(* IEC 61131-3 sources: PortalRobot/Portal_robot/Device/application (part 2) *)

(* ---- FB_MACHINE.st ---- *)
FUNCTION_BLOCK FB_MACHINE
VAR_INPUT
	xExecute          : BOOL; // Запуск разрешённой операции обслуживания
    xReset            : BOOL; // Сброс ошибки конкретного станка
	xResetGlobal      : BOOL; // Общий сброс ошибок ячейки
	xGlobalError      : BOOL; // Глобальная ошибка ячейки
	xHmiSetPartLoaded : BOOL; // Ручное подтверждение загруженной детали
    xHmiSetPartEmpty  : BOOL; // Ручное подтверждение пустого патрона
	xHmiEnable        : BOOL; // Импульс включения станка в работу
	xHmiDisable       : BOOL; // Импульс отключения станка от работы
	stChangeRecipe    : ARRAY [0..40] OF ST_MACHINE_RECIPE; // Рецепт смены детали
	stLoadRecipe      : ARRAY [0..40] OF ST_MACHINE_RECIPE; // Рецепт загрузки заготовки
	stUnloadRecipe    : ARRAY [0..40] OF ST_MACHINE_RECIPE; // Рецепт выгрузки детали
	stPoints          : ST_MACHINE_POINTS; // Имена рабочих точек станка
	stRobotStatus     : ST_ROBOT_STATUS; // Статусы робота
	stMachineStatus   : ST_MACHINE_IO_STATUS; // Состояние исполнительных механизмов станка
END_VAR
VAR_OUTPUT
	Command : ST_MACHINE_COMMAND; // Команды станку и роботу
	Status  : ST_MACHINE_PUBLIC; // Публичные статусы станка
	Diag    : ST_MACHINE_DIAG; // Состояние автомата и выбранная операция
	Error   : ST_MACHINE_ERRORS; // Активные и последние ошибки
END_VAR
VAR
	eState                  : E_MACHINE_STATE := E_MACHINE_STATE.DISABLED; // Текущее состояние автомата
	ePartState              : E_PART_STATE := E_PART_STATE.UNKNOWN; // Состояние детали в патроне
	uiIndex                 : UINT; // Индекс команды рецепта
	tofErrorDoor            : TOF; // Контроль закрытия двери при нахождении робота внутри
	rtExectue               : R_TRIG; // Фронт команды запуска
	rtEnabledMachine        : R_TRIG; // Фронт команды включения
	rtDisabledMachine       : R_TRIG; // Фронт команды отключения
	rtCycleDone             : R_TRIG; // Фронт завершения цикла станка
    rtSetPartLoaded         : R_TRIG; // Фронт ручного подтверждения детали
    rtSetPartEmpty          : R_TRIG; // Фронт ручного подтверждения пустого патрона
	xRetreatStarted         : BOOL; // Начат отход робота от станка
	xRobotInsideMachine     : BOOL; // Робот находится внутри рабочей зоны
	xRobotDone              : BOOL; // Робот освобождён алгоритмом станка
	xServiceDoorCloseDemand : BOOL; // Внутренний запрос закрытия двери
	xServiceDoorOpenDemand  : BOOL; // Внутренний запрос открытия двери
	xAutoDoorOpenLatched    : BOOL; // Защёлка автоматического открытия двери
	eGrantedOperation       : E_MACHINE_OPERATION; // Разрешённая операция обслуживания
	eActualOperation        : E_MACHINE_OPERATION; // Выполняемая операция обслуживания
	stRecipe                : ARRAY [0..40] OF ST_MACHINE_RECIPE; // Активный рецепт операции
END_VAR

VAR CONSTANT
	ERR_WRONG_OPERATION     : DWORD := 1;   	// Приводит к глоабльной ошибке
    ERR_WRONG_COMMAND       : DWORD := 2;   	// Приводит к глобальной ошибке
    ERR_ROBOT_MOTION        : DWORD := 4;   	// Приводит к глобальной ошибке (Другой блок не создаём новую ошибку)
    ERR_ROBOT_ACTION        : DWORD := 8;   	// Приводит к глобальной ошибке (Другой блок не создаём новую ошибку)
    ERR_DOOR_OPEN  			: DWORD := 16;  	// Не приводит к глобальной ошибке, уезжаем в другой станок
	ERR_DOOR_CLOSE 			: DWORD := 32;  	// Не приводит к глобальной ошибке, уезжаем в другой станок
	ERR_CHUCK_OPEN 			: DWORD := 64;  	// Приводит к глобальной ошибке
	ERR_CHUCK_CLOSE 		: DWORD := 128; 	// Приводит к глобальной ошибке
	ERR_CYCLE_START			: DWORD := 256;     // Не приводит к глобальной ошибке
	ERR_SAFETY_STOP         : DWORD := 512;		// Глобальная ошибка из вне (Другой блок не создаём новую ошибку)
	ERR_UNKNOWN_DETAIL      : DWORD := 1024;    // Приводит к глобальной ошибке
	ERR_MACHINE_ALARM       : DWORD := 2048;    // Приводит к глобальной ошибке
	ERR_INDEX               : DWORD := 4096;    // Приводит к глобальной ошибке
	ERR_DOOR_ROBOT          : DWORD := 8192;    // Приводит к глобальной ошибке
	ERR_MACHINE_IDLE        : DWORD := 16384;   // Не приводит к глобальной ошибке

	// Ошибки, требующие формирования глобальной аварии ячейки.
	MASK_CRITICAL_ERROR		: DWORD :=
								ERR_WRONG_OPERATION OR
								ERR_WRONG_COMMAND OR
								ERR_CHUCK_OPEN OR
								ERR_CHUCK_CLOSE OR
								ERR_UNKNOWN_DETAIL OR
								ERR_MACHINE_ALARM OR
								ERR_INDEX OR
								ERR_DOOR_ROBOT;

	// Некритические ошибки конкретного станка.
	MASK_ALARM_ERROR		: DWORD :=
								ERR_DOOR_OPEN OR
								ERR_DOOR_CLOSE OR
								ERR_CYCLE_START OR
								ERR_MACHINE_IDLE;

	// Ошибки, полученные от других блоков или общей логики ячейки.
	MASK_EXTERNAL_ERROR  	: DWORD :=
								ERR_SAFETY_STOP OR
								ERR_ROBOT_ACTION OR
								ERR_ROBOT_MOTION;

END_VAR

// --- BEGIN IMPLEMENTATION ---

(*
	1. Добавить таймауты (использовать уже существующие ошибки)
*)

rtEnabledMachine (CLK :=xHmiEnable);
rtDisabledMachine (CLK :=xHmiDisable);
rtCycleDone(CLK := stMachineStatus.xCycleDone);
rtSetPartLoaded(CLK := xHmiSetPartLoaded);
rtSetPartEmpty(CLK := xHmiSetPartEmpty);

// Команды по умолчанию
Command.stIo.xOpenDoor := FALSE;
Command.stIo.xCloseDoor := FALSE;
Command.stIo.xClampChuck := FALSE;
Command.stIo.xUnclampChuck := FALSE;
Command.stIo.xStartCycle := FALSE;
Command.stIo.xReset := xReset OR xResetGlobal;

Command.stRobot.xExecute := FALSE;
Command.stRobot.xStop := FALSE;
Command.stRobot.eAction := E_ROBOT_ACTION.NONE;
xServiceDoorOpenDemand := FALSE;
xServiceDoorCloseDemand := FALSE;

IF stMachineStatus.xChuckClamped AND NOT stMachineStatus.xAlarm THEN
	ePartState := E_PART_STATE.LOADED;
ELSIF stMachineStatus.xChuckUnclamped AND NOT stMachineStatus.xAlarm THEN
	ePartState := E_PART_STATE.EMPTY;
ELSE
	ePartState := E_PART_STATE.UNKNOWN;
END_IF

// // Ручное подтверждение состояния детали
// IF (eState = E_MACHINE_STATE.IDLE)
// AND NOT stMachineStatus.xCycleActive THEN
//     IF rtSetPartLoaded.Q THEN
//         ePartState := E_PART_STATE.LOADED;
//     END_IF;
//
//     IF rtSetPartEmpty.Q THEN
//         ePartState := E_PART_STATE.EMPTY;
//     END_IF;
// END_IF;

// Автоматическое открытие после окончания обработки
IF rtCycleDone.Q
	AND NOT stMachineStatus.xAlarm
	AND NOT stMachineStatus.xCycleActive
	AND (eState = E_MACHINE_STATE.IDLE)
	AND NOT xGlobalError THEN
    xAutoDoorOpenLatched := TRUE;
END_IF;

IF stMachineStatus.xDoorOpen THEN
    xAutoDoorOpenLatched := FALSE;
END_IF;

IF (ePartState = E_PART_STATE.EMPTY)
AND stRobotStatus.xBlankAvailable THEN
    eGrantedOperation := E_MACHINE_OPERATION.LOAD;

ELSIF (ePartState = E_PART_STATE.LOADED) THEN
    IF stRobotStatus.xBlankAvailable THEN
        eGrantedOperation := E_MACHINE_OPERATION.CHANGE;
    ELSE
        eGrantedOperation := E_MACHINE_OPERATION.UNLOAD;
    END_IF;
ELSIF (ePartState = E_PART_STATE.UNKNOWN) THEN
	eGrantedOperation := E_MACHINE_OPERATION.NONE;
END_IF;

// Включение и отключение блока
IF rtDisabledMachine.Q AND (eState = E_MACHINE_STATE.IDLE) THEN
    eState := E_MACHINE_STATE.DISABLED;
ELSIF rtEnabledMachine.Q AND eState = E_MACHINE_STATE.DISABLED AND NOT stMachineStatus.xAlarm THEN
    eState := E_MACHINE_STATE.IDLE;
ELSIF rtEnabledMachine.Q AND eState = E_MACHINE_STATE.DISABLED AND stMachineStatus.xAlarm THEN
	eState := E_MACHINE_STATE.ERROR;
END_IF;

IF xGlobalError
AND (eState <> E_MACHINE_STATE.IDLE)
AND (eState <> E_MACHINE_STATE.DISABLED)
AND (eState <> E_MACHINE_STATE.ERROR) THEN
    Error.dwErrorActive := Error.dwErrorActive OR ERR_SAFETY_STOP;
    eState := E_MACHINE_STATE.ERROR;
END_IF;

IF stMachineStatus.xAlarm AND (eState = E_MACHINE_STATE.IDLE) THEN
	Error.dwErrorActive := Error.dwErrorActive OR ERR_MACHINE_IDLE;
    eState := E_MACHINE_STATE.ERROR;
END_IF

//Останавливаем робота, если кто-то попытался закрыть дверь в станке в момент его работы
tofErrorDoor(
			PT:= T#100MS,
			IN:=stMachineStatus.xDoorOpen
);

xRobotInsideMachine := (eState = E_MACHINE_STATE.ROBOT_ACTION)
						OR (eState = E_MACHINE_STATE.ROBOT_MOVE)
						OR (eState = E_MACHINE_STATE.RELEASE_ROBOT_ACTION);

IF xRobotInsideMachine AND NOT tofErrorDoor.Q THEN
	Command.stRobot.xStop := TRUE;
	Error.dwErrorActive := Error.dwErrorActive OR ERR_DOOR_ROBOT;
    eState := E_MACHINE_STATE.ERROR;
END_IF

CASE eState OF
	E_MACHINE_STATE.DISABLED:
	;
	E_MACHINE_STATE.IDLE:
		uiIndex := 0;
		xRobotDone := FALSE;
		IF xExecute THEN
			IF (stRobotStatus.eCurrentPoint = stPoints.eAbove)
			AND ePartState <> E_PART_STATE.UNKNOWN
			AND NOT stMachineStatus.xAlarm
			AND NOT stMachineStatus.xCycleActive
    		AND NOT stRobotStatus.xBusy
			AND NOT stRobotStatus.xError
			AND NOT xGlobalError THEN
				eActualOperation := eGrantedOperation;
				eState := E_MACHINE_STATE.CHOSE;
			ELSIF ePartState = E_PART_STATE.UNKNOWN THEN
				Error.dwErrorActive := Error.dwErrorActive OR ERR_UNKNOWN_DETAIL;
				eState := E_MACHINE_STATE.ERROR ;
			END_IF
		END_IF

	E_MACHINE_STATE.CHOSE:
		CASE eActualOperation OF
			E_MACHINE_OPERATION.CHANGE:
				stRecipe := stChangeRecipe;
				eState := E_MACHINE_STATE.READ;
			E_MACHINE_OPERATION.LOAD:
				stRecipe := stLoadRecipe;
				eState := E_MACHINE_STATE.READ;
			E_MACHINE_OPERATION.UNLOAD:
				stRecipe := stUnloadRecipe;
				eState := E_MACHINE_STATE.READ;
		ELSE
			Error.dwErrorActive := Error.dwErrorActive OR ERR_WRONG_OPERATION ;
			eState := E_MACHINE_STATE.ERROR;
		END_CASE

	E_MACHINE_STATE.READ:
		CASE stRecipe[uiIndex].eCommand OF
			E_MACHINE_STATE.ROBOT_MOVE:
				eState := E_MACHINE_STATE.ROBOT_MOVE;

			E_MACHINE_STATE.ROBOT_ACTION:
				eState := E_MACHINE_STATE.ROBOT_ACTION;

			E_MACHINE_STATE.DOOR_OPEN:
				eState := E_MACHINE_STATE.DOOR_OPEN;

			E_MACHINE_STATE.DOOR_CLOSE:
				eState := E_MACHINE_STATE.DOOR_CLOSE;

			E_MACHINE_STATE.CHUCK_OPEN:
				eState := E_MACHINE_STATE.CHUCK_OPEN;

			E_MACHINE_STATE.CHUCK_CLOSE:
				eState := E_MACHINE_STATE.CHUCK_CLOSE;

			E_MACHINE_STATE.CYCLE_START:
				eState := E_MACHINE_STATE.CYCLE_START;

			E_MACHINE_STATE.DONE:
				eState := E_MACHINE_STATE.DONE;

		ELSE
			Error.dwErrorActive := Error.dwErrorActive OR ERR_WRONG_COMMAND;
			eState := E_MACHINE_STATE.ERROR;
		END_CASE

	E_MACHINE_STATE.NEXT:
			uiIndex := uiIndex + 1;
			IF uiIndex > 40 THEN
				Error.dwErrorActive := Error.dwErrorActive OR ERR_INDEX;
				eState := E_MACHINE_STATE.ERROR;
			ELSE
				eState := E_MACHINE_STATE.READ;
			END_IF;

	E_MACHINE_STATE.ROBOT_MOVE:
		Command.stRobot.xExecute  := TRUE;
		Command.stRobot.eAction   := E_ROBOT_ACTION.MOVE_TO_POINT;
		xRetreatStarted          := stRecipe[uiIndex].xRetreatStarted;
		IF stRecipe[uiIndex].stPoint = E_MACHINE_POINTS.ABOVE  THEN
			Command.stRobot.eSetPoint := stPoints.eAbove;
		ELSIF stRecipe[uiIndex].stPoint = E_MACHINE_POINTS.CHUCK THEN
			Command.stRobot.eSetPoint := stPoints.eChuck;
		ELSIF stRecipe[uiIndex].stPoint = E_MACHINE_POINTS.CHUCK_APPROACH THEN
			Command.stRobot.eSetPoint := stPoints.eChuckApproach;
		ELSIF stRecipe[uiIndex].stPoint = E_MACHINE_POINTS.INSIDE THEN
			Command.stRobot.eSetPoint := stPoints.eInside;
		END_IF

		IF stRobotStatus.xError THEN
			Error.dwErrorActive := Error.dwErrorActive OR ERR_ROBOT_MOTION;
			eState := E_MACHINE_STATE.ERROR ;

		ELSIF stMachineStatus.xAlarm THEN
			Command.stRobot.xStop := TRUE;
			Error.dwErrorActive := Error.dwErrorActive OR ERR_MACHINE_ALARM;
			eState := E_MACHINE_STATE.ERROR ;

		ELSIF stRobotStatus.xDone THEN
        	eState := E_MACHINE_STATE.RELEASE_ROBOT_ACTION;

    	END_IF;

	E_MACHINE_STATE.ROBOT_ACTION:
		Command.stRobot.xExecute  := TRUE;
		Command.stRobot.eAction   := stRecipe[uiIndex].eRobotAction;

		IF stMachineStatus.xAlarm THEN
			Command.stRobot.xStop := TRUE;
			Error.dwErrorActive := Error.dwErrorActive OR ERR_MACHINE_ALARM;
			eState := E_MACHINE_STATE.ERROR ;

		ELSIF stRobotStatus.xError THEN
			Error.dwErrorActive := Error.dwErrorActive OR ERR_ROBOT_ACTION;
			eState := E_MACHINE_STATE.ERROR ;

		ELSIF stRobotStatus.xDone THEN
        	eState := E_MACHINE_STATE.RELEASE_ROBOT_ACTION;
    	END_IF;

	E_MACHINE_STATE.RELEASE_ROBOT_ACTION:
		IF NOT stRobotStatus.xBusy
    	AND NOT stRobotStatus.xDone
		AND NOT stRobotStatus.xError THEN
			xRobotDone := stRecipe[uiIndex].xRobotDone;
        	eState := E_MACHINE_STATE.NEXT;

		ELSIF stRobotStatus.xError AND  stRecipe[uiIndex].eRobotAction = E_ROBOT_ACTION.MOVE_TO_POINT THEN
			Error.dwErrorActive := Error.dwErrorActive OR ERR_ROBOT_MOTION;
			eState := E_MACHINE_STATE.ERROR;

		ELSIF stRobotStatus.xError THEN
			Error.dwErrorActive := Error.dwErrorActive OR ERR_ROBOT_ACTION;
			eState := E_MACHINE_STATE.ERROR;
    	END_IF;

	E_MACHINE_STATE.DOOR_OPEN:
		xServiceDoorOpenDemand := TRUE;

    	IF stMachineStatus.xDoorOpen
    	AND NOT stMachineStatus.xAlarm THEN
			xServiceDoorOpenDemand := FALSE;
        	eState := E_MACHINE_STATE.NEXT;
		ELSIF stMachineStatus.xAlarm THEN
			Error.dwErrorActive := Error.dwErrorActive OR ERR_DOOR_OPEN;
			eState := E_MACHINE_STATE.ERROR;
    	END_IF;

	E_MACHINE_STATE.DOOR_CLOSE:
		xServiceDoorCloseDemand := TRUE;

    	IF stMachineStatus.xDoorClosed
    	AND NOT stMachineStatus.xAlarm THEN
			xServiceDoorCloseDemand := FALSE;
        	eState := E_MACHINE_STATE.NEXT;
		ELSIF stMachineStatus.xAlarm THEN
			Error.dwErrorActive := Error.dwErrorActive OR ERR_DOOR_CLOSE;
			eState := E_MACHINE_STATE.ERROR;
    	END_IF;

	E_MACHINE_STATE.CHUCK_OPEN:
		Command.stIo.xUnclampChuck := TRUE;

    	IF stMachineStatus.xChuckUnclamped
		AND NOT stMachineStatus.xAlarm  THEN
			Command.stIo.xUnclampChuck := FALSE;
       		eState := E_MACHINE_STATE.NEXT;
		ELSIF stMachineStatus.xAlarm THEN
			Command.stIo.xUnclampChuck := FALSE;
			Error.dwErrorActive := Error.dwErrorActive OR ERR_CHUCK_OPEN;
			eState := E_MACHINE_STATE.ERROR;
    	END_IF;

	E_MACHINE_STATE.CHUCK_CLOSE:
		Command.stIo.xClampChuck := TRUE;

    	IF stMachineStatus.xChuckClamped
		AND NOT stMachineStatus.xAlarm  THEN
			Command.stIo.xClampChuck := FALSE;
       		eState := E_MACHINE_STATE.NEXT;
		ELSIF stMachineStatus.xAlarm THEN
			Command.stIo.xClampChuck := FALSE;
			Error.dwErrorActive := Error.dwErrorActive OR ERR_CHUCK_CLOSE;
			eState := E_MACHINE_STATE.ERROR;
    	END_IF;

	E_MACHINE_STATE.CYCLE_START:
		IF stMachineStatus.xChuckClamped
    	AND stMachineStatus.xDoorClosed THEN
		Command.stIo.xStartCycle := TRUE;
		END_IF;

        IF stMachineStatus.xCycleActive AND NOT stMachineStatus.xAlarm THEN
			Command.stIo.xStartCycle := FALSE;
            eState := E_MACHINE_STATE.NEXT;
		ELSIF stMachineStatus.xAlarm THEN
			Command.stIo.xStartCycle := FALSE;
			Error.dwErrorActive := Error.dwErrorActive OR ERR_CHUCK_CLOSE;
			eState := E_MACHINE_STATE.ERROR;
        END_IF;

	E_MACHINE_STATE.DONE:
		CASE eActualOperation OF
			E_MACHINE_OPERATION.CHANGE, E_MACHINE_OPERATION.LOAD:
				eActualOperation := E_MACHINE_OPERATION.NONE;
				ePartState := E_PART_STATE.LOADED;
			E_MACHINE_OPERATION.UNLOAD:
				eActualOperation := E_MACHINE_OPERATION.NONE;
				ePartState := E_PART_STATE.EMPTY;
		END_CASE

		IF NOT xExecute THEN
			xRobotDone := FALSE;
			eState := E_MACHINE_STATE.IDLE;
		END_IF

    E_MACHINE_STATE.ERROR:
		uiIndex := 0;
		eActualOperation := E_MACHINE_OPERATION.NONE;
		eGrantedOperation := E_MACHINE_OPERATION.NONE;

    	IF (xReset OR xResetGlobal)
    	AND NOT xGlobalError
    	AND NOT xExecute
		AND NOT stMachineStatus.xAlarm THEN
			Error.dwErrorLast := Error.dwErrorActive;
			Error.dwErrorActive := DWORD#0;
        	eState := E_MACHINE_STATE.DISABLED;
    	END_IF;
END_CASE;

IF (eState <> E_MACHINE_STATE.ERROR)
AND NOT xGlobalError THEN
    IF xServiceDoorCloseDemand
	AND NOT (xAutoDoorOpenLatched OR xServiceDoorOpenDemand)
	AND NOT stMachineStatus.xAlarm THEN
        Command.stIo.xCloseDoor := TRUE;

    ELSIF (xAutoDoorOpenLatched OR xServiceDoorOpenDemand)
	AND NOT xServiceDoorCloseDemand
    AND NOT stMachineStatus.xCycleActive
    AND NOT stMachineStatus.xAlarm THEN
        Command.stIo.xOpenDoor := TRUE;
    END_IF;
END_IF;

Status.xCanAcceptService := (eState = E_MACHINE_STATE.IDLE)
			AND (stRobotStatus.eCurrentPoint = stPoints.eAbove)
			AND ePartState <> E_PART_STATE.UNKNOWN
			AND NOT stMachineStatus.xAlarm
			AND NOT stMachineStatus.xCycleActive
    		AND NOT stRobotStatus.xBusy
			AND NOT stRobotStatus.xError
			AND NOT xGlobalError;

Status.xProcessing := stMachineStatus.xCycleActive;
Status.xPartReady := stMachineStatus.xCycleDone;
Status.xServiceRequired := (eGrantedOperation <> E_MACHINE_OPERATION.NONE)
	AND (eState = E_MACHINE_STATE.IDLE);
Status.xRobotReleased := xRobotDone;
Status.xDone := (eState = E_MACHINE_STATE.DONE);
Status.xBusy := (eState <> E_MACHINE_STATE.IDLE)
    AND (eState <> E_MACHINE_STATE.DISABLED)
    AND (eState <> E_MACHINE_STATE.ERROR)
	AND (eState <> E_MACHINE_STATE.DONE);
Status.xError := (eState = E_MACHINE_STATE.ERROR);
Status.xCriticalError := (Error.dwErrorActive AND MASK_CRITICAL_ERROR) <> DWORD#0;
Status.xAlarmError    := (Error.dwErrorActive AND MASK_ALARM_ERROR) <> DWORD#0;
Status.xExternalError := (Error.dwErrorActive AND MASK_EXTERNAL_ERROR) <> DWORD#0;
Status.xDoorOpen := stMachineStatus.xDoorOpen;
Status.xAlarm := stMachineStatus.xAlarm;
Status.eRecommendedOperation := eGrantedOperation;
Status.ePartState := ePartState;
Status.eAbovePoint := stPoints.eAbove;

Diag.eState := eState;
Diag.eGrantedOperation := eGrantedOperation;
Diag.eActualOperation := eActualOperation;

IF Error.dwErrorActive <> DWORD#0 THEN
	Error.dwErrorLast := Error.dwErrorActive;
END_IF;

Error.stErrorActive := UpdateErrorView(dwError := Error.dwErrorActive);
Error.stErrorLast := UpdateErrorView(dwError := Error.dwErrorLast);

(* ---- FB_MACHINE_SIMULATION.st ---- *)
FUNCTION_BLOCK FB_MACHINE_SIMULATION
VAR_INPUT
    Command : ST_MACHINE_IO_COMMAND; // Команды исполнительным механизмам

    xSimMachineAlarm : BOOL; // Имитация общей аварии станка
    xSimDoorFault    : BOOL; // Имитация неисправности двери
    xSimChuckFault   : BOOL; // Имитация неисправности патрона

    tDoorTime  : TIME := T#5S; // Время открытия или закрытия двери
    tChuckTime : TIME := T#3S; // Время зажима или разжима патрона
    tCycleTime : TIME := T#60S; // Время цикла обработки
END_VAR

VAR_OUTPUT
    Status : ST_MACHINE_IO_STATUS; // Состояние исполнительных механизмов
	Diag   : ST_MACHINE_SIM_DIAG; // Текущие действия симулятора
	Error  : ST_MACHINE_SIM_ERRORS; // Активные и последние ошибки
END_VAR
VAR CONSTANT
	ERR_MACHINE_ALARM : DWORD := DWORD#16#0000_0001; // Авария станка
	ERR_DOOR_FAULT    : DWORD := DWORD#16#0000_0002; // Ошибка двери
	ERR_CHUCK_FAULT   : DWORD := DWORD#16#0000_0004; // Ошибка патрона
END_VAR

VAR
    rtStartCycle : R_TRIG; // Фронт команды запуска цикла

    tonDoorOpen   : TON; // Таймер открытия двери
    tonDoorClose  : TON; // Таймер закрытия двери
    tonChuckClamp : TON; // Таймер зажима патрона
    tonChuckOpen  : TON; // Таймер разжима патрона
    tonCycleStart : TON; // Таймер подтверждения запуска цикла
    tonCycle      : TON; // Таймер обработки

    xDoorOpening   : BOOL; // Выполняется открытие двери
    xDoorClosing   : BOOL; // Выполняется закрытие двери
    xChuckClamping : BOOL; // Выполняется зажим патрона
    xChuckOpening  : BOOL; // Выполняется разжим патрона
    xCycleStarting : BOOL; // Выполняется запуск цикла

    xAlarmLatched : BOOL; // Защёлкнутая авария симулятора
    xInitialized  : BOOL; // Начальные состояния установлены
END_VAR

// --- BEGIN IMPLEMENTATION ---

// =====================================================
// Первичная инициализация
// =====================================================

IF NOT xInitialized THEN
    Status.xDoorOpen := FALSE;
    Status.xDoorClosed := TRUE;

    Status.xChuckClamped := TRUE;
    Status.xChuckUnclamped := FALSE;

    Status.xCycleActive := FALSE;
    Status.xCycleDone := FALSE;
    Status.xAlarm := FALSE;

    xInitialized := TRUE;
END_IF;

// =====================================================
// Детектор запуска цикла
// =====================================================

rtStartCycle(CLK := Command.xStartCycle);

// =====================================================
// Формирование и сброс аварии
// =====================================================

IF xSimMachineAlarm THEN
	Error.dwErrorActive := Error.dwErrorActive OR ERR_MACHINE_ALARM;
END_IF;

IF xSimDoorFault
AND (xDoorOpening OR xDoorClosing) THEN
	Error.dwErrorActive := Error.dwErrorActive OR ERR_DOOR_FAULT;
END_IF;

IF xSimChuckFault
AND (xChuckClamping OR xChuckOpening) THEN
	Error.dwErrorActive := Error.dwErrorActive OR ERR_CHUCK_FAULT;
END_IF;

IF Command.xReset
AND NOT xSimMachineAlarm
AND NOT xSimDoorFault
AND NOT xSimChuckFault THEN
	Error.dwErrorLast := Error.dwErrorActive;
	Error.dwErrorActive := DWORD#0;
END_IF;

xAlarmLatched := Error.dwErrorActive <> DWORD#0;

// =====================================================
// Приём команд станка
// =====================================================

IF NOT xAlarmLatched THEN

    // Открытие двери
    IF Command.xOpenDoor
    AND NOT Status.xDoorOpen
    AND NOT Status.xCycleActive THEN
        xDoorOpening := TRUE;
        xDoorClosing := FALSE;
    END_IF;

    // Закрытие двери
    IF Command.xCloseDoor
    AND NOT Status.xDoorClosed THEN
        xDoorClosing := TRUE;
        xDoorOpening := FALSE;
    END_IF;

    // Зажим патрона
    IF Command.xClampChuck
    AND NOT Status.xChuckClamped
    AND NOT Status.xCycleActive THEN
        xChuckClamping := TRUE;
        xChuckOpening := FALSE;
    END_IF;

    // Разжим патрона
    IF Command.xUnclampChuck
    AND NOT Status.xChuckUnclamped
    AND NOT Status.xCycleActive THEN
        xChuckOpening := TRUE;
        xChuckClamping := FALSE;
    END_IF;

    // Запуск обработки
    IF rtStartCycle.Q
    AND Status.xDoorClosed
    AND Status.xChuckClamped
    AND NOT Status.xCycleActive THEN
        xCycleStarting := TRUE;
        Status.xCycleDone := FALSE;
    END_IF;

END_IF;

// =====================================================
// Таймеры механизмов
// =====================================================

tonDoorOpen(
    IN := xDoorOpening AND NOT xSimDoorFault,
    PT := tDoorTime
);

tonDoorClose(
    IN := xDoorClosing AND NOT xSimDoorFault,
    PT := tDoorTime
);

tonChuckClamp(
    IN := xChuckClamping AND NOT xSimChuckFault,
    PT := tChuckTime
);

tonChuckOpen(
    IN := xChuckOpening AND NOT xSimChuckFault,
    PT := tChuckTime
);

tonCycleStart(
    IN := xCycleStarting,
    PT := T#200MS
);

tonCycle(
    IN := Status.xCycleActive AND NOT xAlarmLatched,
    PT := tCycleTime
);

// =====================================================
// Завершение открытия двери
// =====================================================

IF tonDoorOpen.Q THEN
    Status.xDoorOpen := TRUE;
    Status.xDoorClosed := FALSE;

    xDoorOpening := FALSE;
END_IF;

// =====================================================
// Завершение закрытия двери
// =====================================================

IF tonDoorClose.Q THEN
    Status.xDoorClosed := TRUE;
    Status.xDoorOpen := FALSE;

    xDoorClosing := FALSE;
END_IF;

// =====================================================
// Завершение зажима патрона
// =====================================================

IF tonChuckClamp.Q THEN
    Status.xChuckClamped := TRUE;
    Status.xChuckUnclamped := FALSE;

    xChuckClamping := FALSE;
END_IF;

// =====================================================
// Завершение разжима патрона
// =====================================================

IF tonChuckOpen.Q THEN
    Status.xChuckUnclamped := TRUE;
    Status.xChuckClamped := FALSE;

    xChuckOpening := FALSE;
END_IF;

// =====================================================
// Запуск цикла
// =====================================================

IF tonCycleStart.Q THEN
    Status.xCycleActive := TRUE;
    xCycleStarting := FALSE;
END_IF;

// =====================================================
// Завершение цикла
// =====================================================

IF tonCycle.Q THEN
    Status.xCycleActive := FALSE;
    Status.xCycleDone := TRUE;
END_IF;

// =====================================================
// Реакция на аварийное состояние
// =====================================================

IF xAlarmLatched THEN
    Status.xCycleActive := FALSE;

    xDoorOpening := FALSE;
    xDoorClosing := FALSE;

    xChuckClamping := FALSE;
    xChuckOpening := FALSE;

    xCycleStarting := FALSE;
END_IF;

// =====================================================
// Выходной статус
// =====================================================

Status.xAlarm := xAlarmLatched;
Status.xReady := NOT xAlarmLatched AND NOT Status.xCycleActive;

Diag.xDoorOpening := xDoorOpening;
Diag.xDoorClosing := xDoorClosing;
Diag.xChuckClamping := xChuckClamping;
Diag.xChuckOpening := xChuckOpening;
Diag.xCycleStarting := xCycleStarting;

IF Error.dwErrorActive <> DWORD#0 THEN
	Error.dwErrorLast := Error.dwErrorActive;
END_IF;

Error.stErrorActive := UpdateErrorView(dwError := Error.dwErrorActive);
Error.stErrorLast := UpdateErrorView(dwError := Error.dwErrorLast);

(* ---- FB_MAGAZINE.st ---- *)
FUNCTION_BLOCK FB_MAGAZINE
VAR_INPUT
	stRobotStatus     : ST_ROBOT_STATUS; // Текущие статусы робота
	stMagazineCommand : ST_MAGAZINE_COMMAND; // Команда магазина от автоматической логики
	stHmiCommand      : ST_ROBOT_COMMAND; // Ручная команда магазина с HMI
	xManual           : BOOL; // Разрешение ручного управления
	xReset            : BOOL; // Сброс ошибок магазина
	xGlobalError      : BOOL; // Глобальная ошибка ячейки
	xMode             : BOOL; // Режим робота: TRUE — Modbus, FALSE — SoftMotion
	xHmiEnable        : BOOL; // Импульс включения магазина с HMI
	xHmiDisable       : BOOL; // Импульс отключения магазина с HMI
	uiRows            : UINT; // Число строк матрицы магазина
	uiColumns         : UINT; // Число столбцов матрицы магазина
	lrPitchX          : LREAL; // Шаг между слотами по оси X
	lrPitchY          : LREAL; // Шаг между слотами по оси Y
	lrSafeZ           : LREAL; // Безопасная координата по оси Z
END_VAR
VAR_OUTPUT
	Command : ST_ROBOT_COMMAND; // Текущая пошаговая команда роботу
	Status  : ST_MAGAZINE_STATUS; // Рабочие статусы магазина
	Diag    : ST_MAGAZINE_DIAG; // Состояние автомата магазина
	Error   : ST_MAGAZINE_ERRORS; // Активные и последние ошибки
END_VAR
VAR_IN_OUT
	stDetail : ARRAY [1..GVL_CELL_SETTINGS.NumberDetail] OF ST_DETAIL; // Содержимое слотов магазина
	stPoint  : ARRAY [0..GVL_POINT.iPointNumber] OF ST_POINT; // Глобальная таблица точек робота
END_VAR
VAR
	eGrantedOperation : E_MAGAZINE_OPERATION; // Доступная операция магазина
	eActualOperation  : E_MAGAZINE_OPERATION; // Выполняемая операция магазина

	rtExecute          : R_TRIG; // Фронт команды запуска
	rtEnable           : R_TRIG; // Фронт команды включения
	rtDisable          : R_TRIG; // Фронт команды отключения

	xExecuteRequest    : BOOL; // Активный запрос выполнения операции
	xResetRequest      : BOOL; // Активный запрос сброса
	xStopRequest       : BOOL; // Активный запрос остановки
	xManualCommand     : BOOL; // Команда получена из ручного интерфейса

	iActiveSlotCount   : SINT; // Число активных слотов выбранной матрицы
	iTakeSlot          : SINT; // Слот выбранной заготовки
	iPutSlot           : SINT; // Выбранный свободный слот
	uiStep             : UINT; // Шаг последовательности робота
	uiIndex            : UINT; // Индекс слота для расчёта координат
	uiRow              : UINT; // Строка выбранного слота
	uiColumn           : UINT; // Столбец выбранного слота

	stTakePoint          : ST_POINT; // Рассчитанная рабочая точка взятия
	stPutPoint           : ST_POINT; // Рассчитанная рабочая точка укладки
	stActiveRobotCommand : ST_ROBOT_COMMAND; // Команда роботу текущего шага
END_VAR
VAR CONSTANT
	ERR_WRONG_OPERATION : DWORD := DWORD#16#0000_0001; // Недопустимая операция магазина
	ERR_NO_BLANK        : DWORD := DWORD#16#0000_0002; // В магазине нет заготовки
	ERR_NO_FREE_SLOT    : DWORD := DWORD#16#0000_0004; // В магазине нет свободного слота
	ERR_INVALID_SLOT    : DWORD := DWORD#16#0000_0008; // Недопустимый номер слота
	ERR_SLOT_CONTENT    : DWORD := DWORD#16#0000_0010; // Содержимое слота не соответствует операции
	ERR_ROBOT           : DWORD := DWORD#16#0000_0020; // Ошибка робота при операции магазина
	ERR_GLOBAL_STOP     : DWORD := DWORD#16#0000_0040; // Остановка по глобальной ошибке
	ERR_GEOMETRY        : DWORD := DWORD#16#0000_0080; // Ошибка параметров матрицы магазина
END_VAR

// --- BEGIN IMPLEMENTATION ---

// Активный размер матрицы может быть меньше полного массива деталей.
IF (uiRows > 0)
AND (uiColumns > 0)
AND ((uiRows * uiColumns) <= SINT_TO_UINT(GVL_CELL_SETTINGS.NumberDetail)) THEN
	iActiveSlotCount := UINT_TO_SINT(uiRows * uiColumns);
ELSE
	iActiveSlotCount := 0;
END_IF;

IF iActiveSlotCount > 0 THEN
	Status.iCurrentBlank := FIND_BLANK(
		stDetail := stDetail,
		iSlotCount := iActiveSlotCount
	);
	Status.iCurrentFreeSlot := FIND_FREE_SLOT(
		stDetail := stDetail,
		iSlotCount := iActiveSlotCount
	);
ELSE
	Status.iCurrentBlank := 0;
	Status.iCurrentFreeSlot := 0;
END_IF;

Status.xOutBlank := Status.iCurrentBlank = 0;
Status.xOutFreeSlot := Status.iCurrentFreeSlot = 0;

// Автоматический выбор доступной операции.
eGrantedOperation := E_MAGAZINE_OPERATION.NONE;

IF NOT Status.xOutBlank
AND NOT stRobotStatus.xBlankAvailable
AND NOT stRobotStatus.xDetailAvailable THEN
	eGrantedOperation := E_MAGAZINE_OPERATION.TAKE;

ELSIF NOT Status.xOutFreeSlot
AND Status.xOutBlank
AND stRobotStatus.xDetailAvailable THEN
	eGrantedOperation := E_MAGAZINE_OPERATION.PUT;

ELSIF NOT Status.xOutFreeSlot
AND NOT Status.xOutBlank
AND stRobotStatus.xDetailAvailable THEN
	eGrantedOperation := E_MAGAZINE_OPERATION.CHANGE;
END_IF;

// Команды магазина с HMI принимаются только в ручном режиме.
xManualCommand := xManual AND (
	(stHmiCommand.eSetPoint = E_POINT_NAME.MAGAZINE_TAKE_DETAIL)
	OR (stHmiCommand.eSetPoint = E_POINT_NAME.MAGAZINE_PUT_DETAIL)
	OR (stHmiCommand.eSetPoint = E_POINT_NAME.MAGAZINE_CHANGE_DETAIL)
);

IF xManual THEN
	IF xManualCommand THEN
		xExecuteRequest := stHmiCommand.xExecute;
		xStopRequest := stHmiCommand.xStop;
	ELSE
		xExecuteRequest := FALSE;
		xStopRequest := FALSE;
	END_IF;
ELSE
	xExecuteRequest := stMagazineCommand.xExecute;
	xStopRequest := stMagazineCommand.xStop;
END_IF;

xResetRequest := xReset;

IF xManual THEN
	rtEnable(CLK := xHmiEnable);
	rtDisable(CLK := xHmiDisable);
ELSE
	rtEnable(CLK := stMagazineCommand.xEnable);
	rtDisable(CLK := stMagazineCommand.xDisable);
END_IF;

rtExecute(CLK := xExecuteRequest);

// Значения команды роботу по умолчанию.
Command.xExecute := FALSE;
Command.xStop := FALSE;
Command.xReset := xResetRequest;
Command.eAction := E_ROBOT_ACTION.NONE;
Command.eSetPoint := E_POINT_NAME.NONE;
Command.iTakeSlot := 0;
Command.iPutSlot := 0;

IF xGlobalError
AND (Diag.eState <> E_MAGAZINE_STATE.DISABLED)
AND (Diag.eState <> E_MAGAZINE_STATE.IDLE)
AND (Diag.eState <> E_MAGAZINE_STATE.ERROR) THEN
	Error.dwErrorActive := Error.dwErrorActive OR ERR_GLOBAL_STOP;
	Diag.eState := E_MAGAZINE_STATE.ERROR;
END_IF;

CASE Diag.eState OF
	E_MAGAZINE_STATE.DISABLED:
		IF rtEnable.Q AND NOT xGlobalError THEN
			Diag.eState := E_MAGAZINE_STATE.IDLE;
		END_IF;

	E_MAGAZINE_STATE.IDLE:
		uiStep := 0;
		eActualOperation := E_MAGAZINE_OPERATION.NONE;

		IF rtDisable.Q THEN
			Diag.eState := E_MAGAZINE_STATE.DISABLED;
		ELSIF xGlobalError THEN
			Error.dwErrorActive := Error.dwErrorActive OR ERR_GLOBAL_STOP;
			Diag.eState := E_MAGAZINE_STATE.ERROR;
		ELSIF rtExecute.Q THEN
			IF xManualCommand THEN
				CASE stHmiCommand.eSetPoint OF
					E_POINT_NAME.MAGAZINE_TAKE_DETAIL:
						eActualOperation := E_MAGAZINE_OPERATION.TAKE;
					E_POINT_NAME.MAGAZINE_PUT_DETAIL:
						eActualOperation := E_MAGAZINE_OPERATION.PUT;
					E_POINT_NAME.MAGAZINE_CHANGE_DETAIL:
						eActualOperation := E_MAGAZINE_OPERATION.CHANGE;
				ELSE
					eActualOperation := E_MAGAZINE_OPERATION.NONE;
				END_CASE;
				iTakeSlot := stHmiCommand.iTakeSlot;
				iPutSlot := stHmiCommand.iPutSlot;
			ELSE
				eActualOperation := eGrantedOperation;
				iTakeSlot := Status.iCurrentBlank;
				iPutSlot := Status.iCurrentFreeSlot;
			END_IF;

			Diag.eState := E_MAGAZINE_STATE.CHOOSE;
		END_IF;

	E_MAGAZINE_STATE.CHOOSE:
		IF (iActiveSlotCount = 0)
		OR (NOT xMode AND (
			((uiColumns > 1) AND (lrPitchX = 0.0))
			OR ((uiRows > 1) AND (lrPitchY = 0.0))
			OR (lrSafeZ = stPoint[E_POINT_NAME.MAGAZINE_DETAIL].Z)
			OR (stPoint[E_POINT_NAME.MAGAZINE_DETAIL].SpeedFactor <= 0.1)
			OR (stPoint[E_POINT_NAME.MAGAZINE_DETAIL].SpeedFactor > 1.0)
		)) THEN
			Error.dwErrorActive := Error.dwErrorActive OR ERR_GEOMETRY;
			Diag.eState := E_MAGAZINE_STATE.ERROR;

		ELSIF eActualOperation = E_MAGAZINE_OPERATION.NONE THEN
			Error.dwErrorActive := Error.dwErrorActive OR ERR_WRONG_OPERATION;
			Diag.eState := E_MAGAZINE_STATE.ERROR;

		ELSIF ((eActualOperation = E_MAGAZINE_OPERATION.TAKE)
			OR (eActualOperation = E_MAGAZINE_OPERATION.CHANGE))
		AND ((iTakeSlot < 1) OR (iTakeSlot > iActiveSlotCount)) THEN
			Error.dwErrorActive := Error.dwErrorActive OR ERR_NO_BLANK OR ERR_INVALID_SLOT;
			Diag.eState := E_MAGAZINE_STATE.ERROR;

		ELSIF ((eActualOperation = E_MAGAZINE_OPERATION.PUT)
			OR (eActualOperation = E_MAGAZINE_OPERATION.CHANGE))
		AND ((iPutSlot < 1) OR (iPutSlot > iActiveSlotCount)) THEN
			Error.dwErrorActive := Error.dwErrorActive OR ERR_NO_FREE_SLOT OR ERR_INVALID_SLOT;
			Diag.eState := E_MAGAZINE_STATE.ERROR;

		ELSIF ((eActualOperation = E_MAGAZINE_OPERATION.TAKE)
			OR (eActualOperation = E_MAGAZINE_OPERATION.CHANGE))
		AND (NOT stDetail[iTakeSlot].xInPosition
			OR (stDetail[iTakeSlot].eDetailType <> E_DETAIL_TYPE.BLANK)) THEN
			Error.dwErrorActive := Error.dwErrorActive OR ERR_SLOT_CONTENT;
			Diag.eState := E_MAGAZINE_STATE.ERROR;

		ELSIF ((eActualOperation = E_MAGAZINE_OPERATION.PUT)
			OR (eActualOperation = E_MAGAZINE_OPERATION.CHANGE))
		AND stDetail[iPutSlot].xInPosition THEN
			Error.dwErrorActive := Error.dwErrorActive OR ERR_SLOT_CONTENT;
			Diag.eState := E_MAGAZINE_STATE.ERROR;

		ELSIF (eActualOperation = E_MAGAZINE_OPERATION.TAKE)
		AND (stRobotStatus.xBlankAvailable OR stRobotStatus.xDetailAvailable) THEN
			Error.dwErrorActive := Error.dwErrorActive OR ERR_WRONG_OPERATION;
			Diag.eState := E_MAGAZINE_STATE.ERROR;

		ELSIF ((eActualOperation = E_MAGAZINE_OPERATION.PUT)
			OR (eActualOperation = E_MAGAZINE_OPERATION.CHANGE))
		AND NOT stRobotStatus.xDetailAvailable THEN
			Error.dwErrorActive := Error.dwErrorActive OR ERR_WRONG_OPERATION;
			Diag.eState := E_MAGAZINE_STATE.ERROR;

		ELSE
			IF (eActualOperation = E_MAGAZINE_OPERATION.TAKE)
			OR (eActualOperation = E_MAGAZINE_OPERATION.CHANGE) THEN
				uiIndex := SINT_TO_UINT(iTakeSlot - 1);
				uiColumn := uiIndex MOD uiColumns;
				uiRow := uiIndex / uiColumns;
				stTakePoint := stPoint[E_POINT_NAME.MAGAZINE_DETAIL];
				stTakePoint.X := stTakePoint.X + UINT_TO_LREAL(uiColumn) * lrPitchX;
				stTakePoint.Y := stTakePoint.Y + UINT_TO_LREAL(uiRow) * lrPitchY;
			END_IF;

			IF (eActualOperation = E_MAGAZINE_OPERATION.PUT)
			OR (eActualOperation = E_MAGAZINE_OPERATION.CHANGE) THEN
				uiIndex := SINT_TO_UINT(iPutSlot - 1);
				uiColumn := uiIndex MOD uiColumns;
				uiRow := uiIndex / uiColumns;
				stPutPoint := stPoint[E_POINT_NAME.MAGAZINE_DETAIL];
				stPutPoint.X := stPutPoint.X + UINT_TO_LREAL(uiColumn) * lrPitchX;
				stPutPoint.Y := stPutPoint.Y + UINT_TO_LREAL(uiRow) * lrPitchY;
			END_IF;

			uiStep := 0;
			Diag.eState := E_MAGAZINE_STATE.PREPARE_STEP;
		END_IF;

	E_MAGAZINE_STATE.PREPARE_STEP:
		stActiveRobotCommand.xExecute := FALSE;
		stActiveRobotCommand.xStop := FALSE;
		stActiveRobotCommand.xReset := xResetRequest;
		stActiveRobotCommand.eAction := E_ROBOT_ACTION.NONE;
		stActiveRobotCommand.eSetPoint := E_POINT_NAME.NONE;
		stActiveRobotCommand.iTakeSlot := iTakeSlot;
		stActiveRobotCommand.iPutSlot := iPutSlot;

		IF xMode THEN
			stActiveRobotCommand.eAction := E_ROBOT_ACTION.MOVE_TO_POINT;
			CASE eActualOperation OF
				E_MAGAZINE_OPERATION.TAKE:
					stActiveRobotCommand.eSetPoint := E_POINT_NAME.MAGAZINE_TAKE_DETAIL;
				E_MAGAZINE_OPERATION.PUT:
					stActiveRobotCommand.eSetPoint := E_POINT_NAME.MAGAZINE_PUT_DETAIL;
				E_MAGAZINE_OPERATION.CHANGE:
					stActiveRobotCommand.eSetPoint := E_POINT_NAME.MAGAZINE_CHANGE_DETAIL;
			END_CASE;
			Diag.eState := E_MAGAZINE_STATE.ROBOT_COMMAND;

		ELSE
			CASE eActualOperation OF
				E_MAGAZINE_OPERATION.TAKE:
					CASE uiStep OF
						0: stActiveRobotCommand.eAction := E_ROBOT_ACTION.ROTATE_TO_BLANK;
						1:
							stPoint[E_POINT_NAME.MAGAZINE_TAKE_DETAIL] := stTakePoint;
							stPoint[E_POINT_NAME.MAGAZINE_TAKE_DETAIL].Z := lrSafeZ;
							stActiveRobotCommand.eAction := E_ROBOT_ACTION.MOVE_TO_POINT;
							stActiveRobotCommand.eSetPoint := E_POINT_NAME.MAGAZINE_TAKE_DETAIL;
						2:
							stPoint[E_POINT_NAME.MAGAZINE_TAKE_DETAIL] := stTakePoint;
							stActiveRobotCommand.eAction := E_ROBOT_ACTION.MOVE_TO_POINT;
							stActiveRobotCommand.eSetPoint := E_POINT_NAME.MAGAZINE_TAKE_DETAIL;
						3: stActiveRobotCommand.eAction := E_ROBOT_ACTION.CLAMP_1;
						4:
							stPoint[E_POINT_NAME.MAGAZINE_TAKE_DETAIL] := stTakePoint;
							stPoint[E_POINT_NAME.MAGAZINE_TAKE_DETAIL].Z := lrSafeZ;
							stActiveRobotCommand.eAction := E_ROBOT_ACTION.MOVE_TO_POINT;
							stActiveRobotCommand.eSetPoint := E_POINT_NAME.MAGAZINE_TAKE_DETAIL;
					ELSE
						Diag.eState := E_MAGAZINE_STATE.DONE;
					END_CASE;

				E_MAGAZINE_OPERATION.PUT:
					CASE uiStep OF
						0: stActiveRobotCommand.eAction := E_ROBOT_ACTION.ROTATE_TO_DETAIL;
						1:
							stPoint[E_POINT_NAME.MAGAZINE_PUT_DETAIL] := stPutPoint;
							stPoint[E_POINT_NAME.MAGAZINE_PUT_DETAIL].Z := lrSafeZ;
							stActiveRobotCommand.eAction := E_ROBOT_ACTION.MOVE_TO_POINT;
							stActiveRobotCommand.eSetPoint := E_POINT_NAME.MAGAZINE_PUT_DETAIL;
						2:
							stPoint[E_POINT_NAME.MAGAZINE_PUT_DETAIL] := stPutPoint;
							stActiveRobotCommand.eAction := E_ROBOT_ACTION.MOVE_TO_POINT;
							stActiveRobotCommand.eSetPoint := E_POINT_NAME.MAGAZINE_PUT_DETAIL;
						3: stActiveRobotCommand.eAction := E_ROBOT_ACTION.UNCLAMP_2;
						4:
							stPoint[E_POINT_NAME.MAGAZINE_PUT_DETAIL] := stPutPoint;
							stPoint[E_POINT_NAME.MAGAZINE_PUT_DETAIL].Z := lrSafeZ;
							stActiveRobotCommand.eAction := E_ROBOT_ACTION.MOVE_TO_POINT;
							stActiveRobotCommand.eSetPoint := E_POINT_NAME.MAGAZINE_PUT_DETAIL;
					ELSE
						Diag.eState := E_MAGAZINE_STATE.DONE;
					END_CASE;

				E_MAGAZINE_OPERATION.CHANGE:
					CASE uiStep OF
						0: stActiveRobotCommand.eAction := E_ROBOT_ACTION.ROTATE_TO_DETAIL;
						1:
							stPoint[E_POINT_NAME.MAGAZINE_PUT_DETAIL] := stPutPoint;
							stPoint[E_POINT_NAME.MAGAZINE_PUT_DETAIL].Z := lrSafeZ;
							stActiveRobotCommand.eAction := E_ROBOT_ACTION.MOVE_TO_POINT;
							stActiveRobotCommand.eSetPoint := E_POINT_NAME.MAGAZINE_PUT_DETAIL;
						2:
							stPoint[E_POINT_NAME.MAGAZINE_PUT_DETAIL] := stPutPoint;
							stActiveRobotCommand.eAction := E_ROBOT_ACTION.MOVE_TO_POINT;
							stActiveRobotCommand.eSetPoint := E_POINT_NAME.MAGAZINE_PUT_DETAIL;
						3: stActiveRobotCommand.eAction := E_ROBOT_ACTION.UNCLAMP_2;
						4:
							stPoint[E_POINT_NAME.MAGAZINE_PUT_DETAIL] := stPutPoint;
							stPoint[E_POINT_NAME.MAGAZINE_PUT_DETAIL].Z := lrSafeZ;
							stActiveRobotCommand.eAction := E_ROBOT_ACTION.MOVE_TO_POINT;
							stActiveRobotCommand.eSetPoint := E_POINT_NAME.MAGAZINE_PUT_DETAIL;
						5: stActiveRobotCommand.eAction := E_ROBOT_ACTION.ROTATE_TO_BLANK;
						6:
							stPoint[E_POINT_NAME.MAGAZINE_TAKE_DETAIL] := stTakePoint;
							stPoint[E_POINT_NAME.MAGAZINE_TAKE_DETAIL].Z := lrSafeZ;
							stActiveRobotCommand.eAction := E_ROBOT_ACTION.MOVE_TO_POINT;
							stActiveRobotCommand.eSetPoint := E_POINT_NAME.MAGAZINE_TAKE_DETAIL;
						7:
							stPoint[E_POINT_NAME.MAGAZINE_TAKE_DETAIL] := stTakePoint;
							stActiveRobotCommand.eAction := E_ROBOT_ACTION.MOVE_TO_POINT;
							stActiveRobotCommand.eSetPoint := E_POINT_NAME.MAGAZINE_TAKE_DETAIL;
						8: stActiveRobotCommand.eAction := E_ROBOT_ACTION.CLAMP_1;
						9:
							stPoint[E_POINT_NAME.MAGAZINE_TAKE_DETAIL] := stTakePoint;
							stPoint[E_POINT_NAME.MAGAZINE_TAKE_DETAIL].Z := lrSafeZ;
							stActiveRobotCommand.eAction := E_ROBOT_ACTION.MOVE_TO_POINT;
							stActiveRobotCommand.eSetPoint := E_POINT_NAME.MAGAZINE_TAKE_DETAIL;
					ELSE
						Diag.eState := E_MAGAZINE_STATE.DONE;
					END_CASE;
			END_CASE;

			IF Diag.eState = E_MAGAZINE_STATE.PREPARE_STEP THEN
				Diag.eState := E_MAGAZINE_STATE.ROBOT_COMMAND;
			END_IF;
		END_IF;

	E_MAGAZINE_STATE.ROBOT_COMMAND:
		Command := stActiveRobotCommand;
		Command.xExecute := TRUE;

		IF xStopRequest OR xGlobalError THEN
			Command.xStop := TRUE;
			Error.dwErrorActive := Error.dwErrorActive OR ERR_GLOBAL_STOP;
			Diag.eState := E_MAGAZINE_STATE.ERROR;

		ELSIF stRobotStatus.xError THEN
			Error.dwErrorActive := Error.dwErrorActive OR ERR_ROBOT;
			Diag.eState := E_MAGAZINE_STATE.ERROR;

		ELSIF stRobotStatus.xDone THEN
			IF xMode THEN
				IF (eActualOperation = E_MAGAZINE_OPERATION.PUT)
				OR (eActualOperation = E_MAGAZINE_OPERATION.CHANGE) THEN
					stDetail[iPutSlot].xInPosition := TRUE;
					stDetail[iPutSlot].eDetailType := E_DETAIL_TYPE.DETAIL;
				END_IF;
				IF (eActualOperation = E_MAGAZINE_OPERATION.TAKE)
				OR (eActualOperation = E_MAGAZINE_OPERATION.CHANGE) THEN
					stDetail[iTakeSlot].xInPosition := FALSE;
					stDetail[iTakeSlot].eDetailType := E_DETAIL_TYPE.NONE;
				END_IF;
			ELSE
				IF (uiStep = 3)
				AND ((eActualOperation = E_MAGAZINE_OPERATION.PUT)
					OR (eActualOperation = E_MAGAZINE_OPERATION.CHANGE)) THEN
					stDetail[iPutSlot].xInPosition := TRUE;
					stDetail[iPutSlot].eDetailType := E_DETAIL_TYPE.DETAIL;
				END_IF;
				IF ((uiStep = 3) AND (eActualOperation = E_MAGAZINE_OPERATION.TAKE))
				OR ((uiStep = 8) AND (eActualOperation = E_MAGAZINE_OPERATION.CHANGE)) THEN
					stDetail[iTakeSlot].xInPosition := FALSE;
					stDetail[iTakeSlot].eDetailType := E_DETAIL_TYPE.NONE;
				END_IF;
			END_IF;

			Diag.eState := E_MAGAZINE_STATE.RELEASE_ROBOT_COMMAND;
		END_IF;

	E_MAGAZINE_STATE.RELEASE_ROBOT_COMMAND:
		IF stRobotStatus.xError THEN
			Error.dwErrorActive := Error.dwErrorActive OR ERR_ROBOT;
			Diag.eState := E_MAGAZINE_STATE.ERROR;
		ELSIF NOT stRobotStatus.xBusy AND NOT stRobotStatus.xDone THEN
			IF xMode THEN
				Diag.eState := E_MAGAZINE_STATE.DONE;
			ELSE
				Diag.eState := E_MAGAZINE_STATE.NEXT;
			END_IF;
		END_IF;

	E_MAGAZINE_STATE.NEXT:
		uiStep := uiStep + 1;
		Diag.eState := E_MAGAZINE_STATE.PREPARE_STEP;

	E_MAGAZINE_STATE.DONE:
		IF NOT xExecuteRequest THEN
			eActualOperation := E_MAGAZINE_OPERATION.NONE;
			Diag.eState := E_MAGAZINE_STATE.IDLE;
		END_IF;

	E_MAGAZINE_STATE.ERROR:
		IF stRobotStatus.xBusy THEN
			Command := stActiveRobotCommand;
			Command.xExecute := TRUE;
			Command.xStop := TRUE;
		END_IF;

		IF xResetRequest
		AND NOT xExecuteRequest
		AND NOT xGlobalError
		AND NOT stRobotStatus.xError THEN
			Error.dwErrorLast := Error.dwErrorActive;
			Error.dwErrorActive := DWORD#0;
			eActualOperation := E_MAGAZINE_OPERATION.NONE;
			Diag.eState := E_MAGAZINE_STATE.DISABLED;
		END_IF;
END_CASE;

Status.xEnabled := Diag.eState <> E_MAGAZINE_STATE.DISABLED;
Status.xReady := Diag.eState = E_MAGAZINE_STATE.IDLE;
Status.xBusy := (Diag.eState <> E_MAGAZINE_STATE.DISABLED)
	AND (Diag.eState <> E_MAGAZINE_STATE.IDLE)
	AND (Diag.eState <> E_MAGAZINE_STATE.DONE)
	AND (Diag.eState <> E_MAGAZINE_STATE.ERROR);
Status.xDone := Diag.eState = E_MAGAZINE_STATE.DONE;
Status.xError := Diag.eState = E_MAGAZINE_STATE.ERROR;
Status.eGrantedOperation := eGrantedOperation;
Status.eActualOperation := eActualOperation;
Status.iSelectedBlank := iTakeSlot;
Status.iSelectedFreeSlot := iPutSlot;
Status.xFinished := Status.xOutBlank
	AND Status.xOutFreeSlot
	AND NOT stRobotStatus.xBlankAvailable
	AND NOT stRobotStatus.xDetailAvailable
	AND NOT Status.xBusy;

IF Error.dwErrorActive <> DWORD#0 THEN
	Error.dwErrorLast := Error.dwErrorActive;
END_IF;

Error.stErrorActive := UpdateErrorView(dwError := Error.dwErrorActive);
Error.stErrorLast := UpdateErrorView(dwError := Error.dwErrorLast);

(* ---- FB_MOTION_MANAGER.st ---- *)
FUNCTION_BLOCK FB_MOTION_MANAGER
VAR_INPUT
	stPoint : ARRAY [0..GVL_POINT.iPointNumber] OF ST_POINT; // Глобальная таблица точек
	xReset  : BOOL; // Сброс ошибок менеджера движения
END_VAR
VAR_OUTPUT
END_VAR
VAR
	curPoint      : ST_POINT; // Координаты выбранной точки
	curPointName  : E_POINT_NAME; // Имя выбранной точки
	fbPointManager: FB_POINT_MANAGER; // Проверка координат и скорости точки
END_VAR
VAR CONSTANT
	ERR_POINT_INVALID : DWORD := DWORD#16#0000_0001; // Недопустимая точка
	ERR_GROUP         : DWORD := DWORD#16#0000_0002; // Ошибка группы осей
	ERR_GLOBAL_STOP   : DWORD := DWORD#16#0000_0004; // Глобальная ошибка ячейки
END_VAR
VAR_IN_OUT
	stMotionManager : ST_MOTION_MANAGER; // Команды, статусы и диагностика менеджера движения
	GroupData       : ST_AXIS_GROUP; // Команды, статусы и диагностика группы XYZ
	stPointManager  : ST_POINT_MANAGER; // Команды, статусы и диагностика проверки точки
END_VAR

// --- BEGIN IMPLEMENTATION ---

stPointManager.Diag.lrX_MinLimit := -1000;
stPointManager.Diag.lrX_MaxLimit := 17000;
stPointManager.Diag.lrY_MinLimit := -1000;
stPointManager.Diag.lrY_MaxLimit := 17000;
stPointManager.Diag.lrZ_MinLimit := -1000;
stPointManager.Diag.lrZ_MaxLimit := 17000;
fbPointManager(
			stPointManager := stPointManager,
			stPoint := curPoint
		);

stMotionManager.Status.xBusy := FALSE;
stMotionManager.Status.xDone := FALSE;
stMotionManager.Status.xError := FALSE;
stMotionManager.Status.xReady:= FALSE;
stMotionManager.Command.xReset := xReset;

CASE stMotionManager.Diag.eState OF
	// --------------------------------------------------
	E_MOTION_MANAGER_STATE.IDLE:
	// --------------------------------------------------
		stMotionManager.Status.xReady:= TRUE;
		IF stMotionManager.Command.xExecute AND NOT stMotionManager.Command.xGlobalError THEN
			stMotionManager.Status.xBusy := TRUE;
			stMotionManager.Diag.eState := E_MOTION_MANAGER_STATE.VALIDATE;
		ELSIF stMotionManager.Command.xGlobalError THEN
			stMotionManager.Error.dwErrorActive := stMotionManager.Error.dwErrorActive OR ERR_GLOBAL_STOP;
			stMotionManager.Diag.eState := E_MOTION_MANAGER_STATE.ERROR;
		END_IF

	// --------------------------------------------------
	E_MOTION_MANAGER_STATE.VALIDATE:
	// --------------------------------------------------
		stMotionManager.Status.xBusy := TRUE;
		curPoint := stPoint[stMotionManager.Command.eTargetPoint];
		curPointName := stMotionManager.Command.eTargetPoint;

		stPointManager.Command.xExecute := TRUE;

		IF stPointManager.Status.xDone AND NOT stPointManager.Status.xInvalid THEN
			stPointManager.Command.xExecute := FALSE;
			IF stMotionManager.Command.xMode THEN
				stMotionManager.Diag.eState := 	E_MOTION_MANAGER_STATE.MOTION_MODBUS;
			ELSE
				stMotionManager.Diag.eState := 	E_MOTION_MANAGER_STATE.MOTION_SIM;
			END_IF
		ELSIF stPointManager.Status.xDone AND stPointManager.Status.xInvalid THEN
			stMotionManager.Error.dwErrorActive := stMotionManager.Error.dwErrorActive OR ERR_POINT_INVALID;
			stMotionManager.Diag.eState := 	E_MOTION_MANAGER_STATE.ERROR;
		END_IF

	// --------------------------------------------------
	E_MOTION_MANAGER_STATE.MOTION_SIM:
	// --------------------------------------------------

		stMotionManager.Status.xBusy := TRUE;

		GroupData.MotionParam.lrX := curPoint.X;
		GroupData.MotionParam.lrY := curPoint.Y;
		GroupData.MotionParam.lrZ := curPoint.Z;
		GroupData.MotionParam.VelFactor := curPoint.SpeedFactor;
		GroupData.MotionParam.AccFactor := curPoint.SpeedFactor;
		GroupData.MotionParam.JerkFactor := curPoint.SpeedFactor;
		IF GroupData.Diag.iStep = E_AXIS_GROUP_STATE.READY AND NOT GroupData.Command.xMoveDirect AND NOT stMotionManager.Command.xGlobalError THEN
			GroupData.Command.xMoveDirect := TRUE;
		END_IF;

		IF GroupData.Status.xMoveDirectDone AND GroupData.Command.xMoveDirect THEN
			GroupData.Command.xMoveDirect := FALSE;
			stMotionManager.Status.eCurrentPoint := curPointName;
			stMotionManager.Diag.eState := 	E_MOTION_MANAGER_STATE.DONE;
		ELSIF GroupData.Diag.iStep = E_AXIS_GROUP_STATE.ERROR OR stMotionManager.Command.xGlobalError  THEN
			IF GroupData.Diag.iStep = E_AXIS_GROUP_STATE.ERROR THEN
				stMotionManager.Error.dwErrorActive := stMotionManager.Error.dwErrorActive OR ERR_GROUP;
			END_IF;
			IF stMotionManager.Command.xGlobalError THEN
				stMotionManager.Error.dwErrorActive := stMotionManager.Error.dwErrorActive OR ERR_GLOBAL_STOP;
			END_IF;
			stMotionManager.Diag.eState := 	E_MOTION_MANAGER_STATE.ERROR;
		END_IF

	// --------------------------------------------------
	E_MOTION_MANAGER_STATE.ERROR:
	// --------------------------------------------------
		stMotionManager.Status.xError := TRUE;
		IF NOT stMotionManager.Command.xGlobalError AND stMotionManager.Command.xReset THEN
			stMotionManager.Error.dwErrorLast := stMotionManager.Error.dwErrorActive;
			stMotionManager.Error.dwErrorActive := DWORD#0;
			stMotionManager.Status.xError := FALSE;
			stMotionManager.Diag.eState := 	E_MOTION_MANAGER_STATE.IDLE;
		END_IF

	// --------------------------------------------------
	E_MOTION_MANAGER_STATE.DONE:
	// --------------------------------------------------
		stMotionManager.Status.xBusy := FALSE;
		stMotionManager.Status.xDone := TRUE;
		IF NOT stMotionManager.Command.xExecute THEN
			stMotionManager.Diag.eState := 	E_MOTION_MANAGER_STATE.IDLE;
		END_IF
	END_CASE

stMotionManager.Error.stErrorActive := UpdateErrorView(
	dwError := stMotionManager.Error.dwErrorActive
);
stMotionManager.Error.stErrorLast := UpdateErrorView(
	dwError := stMotionManager.Error.dwErrorLast
);

(* ---- FB_POINT_MANAGER.st ---- *)
FUNCTION_BLOCK FB_POINT_MANAGER
VAR_INPUT
	stPoint : ST_POINT; // Проверяемая точка
END_VAR
VAR_OUTPUT
END_VAR
VAR
END_VAR
VAR_IN_OUT
	stPointManager : ST_POINT_MANAGER; // Команды, статусы и диагностика проверки точки
END_VAR
VAR CONSTANT
	X_OUT_OF_LIMIT : DWORD := 1; // Координата X вне допустимых границ
	Y_OUT_OF_LIMIT : DWORD := 2; // Координата Y вне допустимых границ
	Z_OUT_OF_LIMIT : DWORD := 4; // Координата Z вне допустимых границ
	INVALID_VEL    : DWORD := 8; // Недопустимый коэффициент скорости
END_VAR

// --- BEGIN IMPLEMENTATION ---

stPointManager.Status.xBusy := FALSE;
stPointManager.Status.xDone := FALSE;
stPointManager.Status.xInvalid := FALSE;

CASE stPointManager.Diag.eState OF
	// --------------------------------------------------
	E_POINT_MANAGER_STATE.IDLE:
	// --------------------------------------------------
		stPointManager.Error.dwErrorActive := DWORD#0;
		IF stPointManager.Command.xExecute THEN
			stPointManager.Status.xBusy := TRUE;
			stPointManager.Diag.eState := E_POINT_MANAGER_STATE.CHECK_ZONE;
		END_IF

	// --------------------------------------------------
	E_POINT_MANAGER_STATE.CHECK_ZONE:
	// --------------------------------------------------
		stPointManager.Status.xBusy := TRUE;

		IF NOT ((stPointManager.Diag.lrX_MinLimit <= stPoint.X) AND (stPoint.X <= stPointManager.Diag.lrX_MaxLimit)) THEN
			stPointManager.Error.dwErrorActive := stPointManager.Error.dwErrorActive OR X_OUT_OF_LIMIT;
		END_IF

		IF NOT ((stPointManager.Diag.lrY_MinLimit <= stPoint.Y) AND (stPoint.Y <= stPointManager.Diag.lrY_MaxLimit)) THEN
			stPointManager.Error.dwErrorActive := stPointManager.Error.dwErrorActive OR Y_OUT_OF_LIMIT;
		END_IF

		IF NOT ((stPointManager.Diag.lrZ_MinLimit <= stPoint.Z) AND (stPoint.Z <= stPointManager.Diag.lrZ_MaxLimit)) THEN
			stPointManager.Error.dwErrorActive := stPointManager.Error.dwErrorActive OR Z_OUT_OF_LIMIT;
		END_IF

		stPointManager.Diag.eState := E_POINT_MANAGER_STATE.CHECK_VEL_FACTOR;

	// --------------------------------------------------
	E_POINT_MANAGER_STATE.CHECK_VEL_FACTOR:
	// --------------------------------------------------
		stPointManager.Status.xBusy := TRUE;

		IF  NOT ((0.1 < stPoint.SpeedFactor) AND(stPoint.SpeedFactor <= 1.0))  THEN
			stPointManager.Error.dwErrorActive := stPointManager.Error.dwErrorActive OR INVALID_VEL;
		END_IF

		stPointManager.Diag.eState := E_POINT_MANAGER_STATE.CHECK_ALL;

	// --------------------------------------------------
	E_POINT_MANAGER_STATE.CHECK_ALL:
	// --------------------------------------------------
		stPointManager.Status.xDone := TRUE;
		stPointManager.Status.xBusy := FALSE;
		IF stPointManager.Error.dwErrorActive <> DWORD#0 THEN
			stPointManager.Status.xInvalid := TRUE;
			stPointManager.Error.dwErrorLast := stPointManager.Error.dwErrorActive;
		ELSE
			stPointManager.Status.xInvalid := FALSE;
		END_IF

		IF NOT stPointManager.Command.xExecute THEN
			stPointManager.Diag.eState := E_POINT_MANAGER_STATE.IDLE;
		END_IF

END_CASE

stPointManager.Error.stErrorActive := UpdateErrorView(
	dwError := stPointManager.Error.dwErrorActive
);
stPointManager.Error.stErrorLast := UpdateErrorView(
	dwError := stPointManager.Error.dwErrorLast
);

(* ---- FB_ROBOT.st ---- *)
FUNCTION_BLOCK FB_ROBOT
VAR_INPUT

	stMachine_1_Command : ST_ROBOT_COMMAND; // Команда роботу от первого станка
	stMachine_2_Command : ST_ROBOT_COMMAND; // Команда роботу от второго станка
	stMachine_3_Command : ST_ROBOT_COMMAND; // Команда роботу от третьего станка
	stMagazineCommand   : ST_ROBOT_COMMAND; // Команда роботу от магазина
	stHmiCommand        : ST_ROBOT_COMMAND; // Ручная команда роботу с HMI
	xReset              : BOOL; // Сброс ошибок робота
    xMode               : BOOL; // Режим робота: TRUE — Modbus, FALSE — SoftMotion
	xManual      		: BOOL; // 1 - ручной режим работы, 0 - автоматический режим работы
	xGlobalError        : BOOL; // Глобальная ошибка ячейки
	xModbusBusy         : BOOL; // Внешний робот выполняет команду
	xModbusDone         : BOOL; // Внешний робот завершил команду
	xModbusError        : BOOL; // Ошибка обмена или внешнего робота

    stPoint : ARRAY [0..GVL_POINT.iPointNumber] OF ST_POINT; // Глобальная таблица точек робота

    xSimBlankAvailable : BOOL; // Начальное наличие заготовки в модели захвата

END_VAR
VAR_OUTPUT
	Command       : ST_ROBOT_COMMAND; // Выбранная команда текущего цикла
	ModbusCommand : ST_ROBOT_COMMAND; // Команда внешнему роботу по Modbus
	Status        : ST_ROBOT_STATUS; // Рабочие статусы робота
	Diag          : ST_ROBOT_DIAG; // Состояние автомата и активная команда
	Error         : ST_ROBOT_ERRORS; // Активные и последние ошибки
END_VAR
VAR
	fbMotionManager  : FB_MOTION_MANAGER; // Менеджер перемещения по точкам
    fbGripper        : FB_GRIPPER_SIMULATION; // Модель двухпозиционного захвата
	stGripperCommand : ST_GRIPPER_COMMAND; // Команда внутренней модели захвата

    eState        : E_ROBOT_STATE := E_ROBOT_STATE.IDLE; // Текущее состояние автомата робота
    eActiveAction : E_ROBOT_ACTION := E_ROBOT_ACTION.NONE; // Защёлкнутое действие
    eActivePoint  : E_POINT_NAME; // Защёлкнутая целевая точка

    xMotionExecute  : BOOL; // Запрос выполнения перемещения
    xGripperExecute : BOOL; // Запрос выполнения действия захвата
	xMagazineCommandActive : BOOL; // Активная команда получена от FB_MAGAZINE

END_VAR

VAR_IN_OUT
    stMotionManager : ST_MOTION_MANAGER; // Данные менеджера движения
    GroupData       : ST_AXIS_GROUP; // Данные группы осей XYZ
    stPointManager  : ST_POINT_MANAGER; // Данные проверки точки
END_VAR

VAR CONSTANT
	ERR_ROBOT_WRONG_ACTION : DWORD := DWORD#16#0000_0001; // Недопустимое действие робота
    ERR_ROBOT_MOTION       : DWORD := DWORD#16#0000_0002; // Ошибка менеджера движения
    ERR_ROBOT_GRIPPER      : DWORD := DWORD#16#0000_0004; // Ошибка захвата
    ERR_ROBOT_MODBUS_STUB  : DWORD := DWORD#16#0000_0008; // Ошибка внешнего робота или Modbus
    ERR_ROBOT_STOP         : DWORD := DWORD#16#0000_0010; // Остановка команды робота
END_VAR

// --- BEGIN IMPLEMENTATION ---

// Команды по умолчанию
xMotionExecute := FALSE;
xGripperExecute := FALSE;
xMagazineCommandActive := FALSE;

Command.xExecute := FALSE;
Command.xStop := FALSE;
Command.xReset := FALSE;
Command.eAction := E_ROBOT_ACTION.NONE;
Command.eSetPoint := E_POINT_NAME.NONE;
Command.iTakeSlot := 0;
Command.iPutSlot := 0;

ModbusCommand.xExecute := FALSE;
ModbusCommand.xStop := FALSE;
ModbusCommand.xReset := xReset;
ModbusCommand.eAction := E_ROBOT_ACTION.NONE;
ModbusCommand.eSetPoint := E_POINT_NAME.NONE;
ModbusCommand.iTakeSlot := 0;
ModbusCommand.iPutSlot := 0;

//Определяем какой режим работы активен
IF NOT xManual THEN
	IF stMachine_1_Command.xExecute THEN
		Command := stMachine_1_Command;
	ELSIF stMachine_2_Command.xExecute THEN
		Command := stMachine_2_Command;
	ELSIF stMachine_3_Command.xExecute THEN
		Command := stMachine_3_Command;
	ELSIF stMagazineCommand.xExecute OR stMagazineCommand.xStop THEN
		Command := stMagazineCommand;
		xMagazineCommandActive := TRUE;
	END_IF
ELSE
	IF stMagazineCommand.xExecute OR stMagazineCommand.xStop THEN
		Command := stMagazineCommand;
		xMagazineCommandActive := TRUE;
	ELSE
		Command := stHmiCommand;
	END_IF
END_IF;

Command.xReset := xReset;

// =====================================================
// Автомат FB_ROBOT
// =====================================================

CASE eState OF

    E_ROBOT_STATE.IDLE:

        Status.xBusy := FALSE;
        Status.xDone := FALSE;
        Status.xError := FALSE;

        IF Command.xExecute
		AND (xMagazineCommandActive
			OR ((Command.eSetPoint <> E_POINT_NAME.MAGAZINE_TAKE_DETAIL)
				AND (Command.eSetPoint <> E_POINT_NAME.MAGAZINE_PUT_DETAIL)
				AND (Command.eSetPoint <> E_POINT_NAME.MAGAZINE_CHANGE_DETAIL))) THEN
            eActiveAction := Command.eAction;
            eActivePoint := Command.eSetPoint;

            IF xMode THEN
                eState := E_ROBOT_STATE.MODBUS_STUB;

            ELSE
                CASE Command.eAction OF

                    E_ROBOT_ACTION.MOVE_TO_POINT:
                        eState := E_ROBOT_STATE.MOTION;

                    E_ROBOT_ACTION.UNCLAMP_1,
                    E_ROBOT_ACTION.CLAMP_1,
                    E_ROBOT_ACTION.UNCLAMP_2,
                    E_ROBOT_ACTION.CLAMP_2,
                    E_ROBOT_ACTION.ROTATE_TO_BLANK,
                    E_ROBOT_ACTION.ROTATE_TO_DETAIL:
                        eState := E_ROBOT_STATE.GRIPPER;

                ELSE
                    Error.dwErrorActive :=
                        Error.dwErrorActive OR ERR_ROBOT_WRONG_ACTION;

                    eState := E_ROBOT_STATE.ERROR;
                END_CASE;
            END_IF;
        END_IF;

    E_ROBOT_STATE.MOTION:

        Status.xBusy := TRUE;
        xMotionExecute := TRUE;

        IF Command.xStop OR xGlobalError THEN
            Error.dwErrorActive := Error.dwErrorActive OR ERR_ROBOT_STOP;
            eState := E_ROBOT_STATE.ERROR;

        ELSIF stMotionManager.Status.xError THEN
            Error.dwErrorActive := Error.dwErrorActive OR ERR_ROBOT_MOTION;
            eState := E_ROBOT_STATE.ERROR;

        ELSIF stMotionManager.Status.xDone THEN
            eState := E_ROBOT_STATE.DONE;
        END_IF;

    E_ROBOT_STATE.GRIPPER:

        Status.xBusy := TRUE;
        xGripperExecute := TRUE;

        IF Command.xStop OR xGlobalError THEN
            Error.dwErrorActive := Error.dwErrorActive OR ERR_ROBOT_STOP;
            eState := E_ROBOT_STATE.ERROR;

        ELSIF fbGripper.Status.xError THEN
            Error.dwErrorActive := Error.dwErrorActive OR ERR_ROBOT_GRIPPER;
            eState := E_ROBOT_STATE.ERROR;

        ELSIF fbGripper.Status.xDone THEN
            eState := E_ROBOT_STATE.DONE;
        END_IF;

    E_ROBOT_STATE.DONE:

        Status.xBusy := FALSE;
        Status.xDone := TRUE;

        CASE eActiveAction OF

            E_ROBOT_ACTION.MOVE_TO_POINT:
                xMotionExecute := TRUE;

            E_ROBOT_ACTION.UNCLAMP_1,
            E_ROBOT_ACTION.CLAMP_1,
            E_ROBOT_ACTION.UNCLAMP_2,
            E_ROBOT_ACTION.CLAMP_2,
            E_ROBOT_ACTION.ROTATE_TO_BLANK,
            E_ROBOT_ACTION.ROTATE_TO_DETAIL:
                xGripperExecute := TRUE;

        END_CASE;

        IF NOT Command.xExecute THEN
            Status.xDone := FALSE;
            eActiveAction := E_ROBOT_ACTION.NONE;
            eState := E_ROBOT_STATE.IDLE;
        END_IF;

    E_ROBOT_STATE.MODBUS_STUB:
		Status.xBusy := TRUE;
		ModbusCommand := Command;
		ModbusCommand.xExecute := TRUE;

		IF Command.xStop OR xGlobalError THEN
			ModbusCommand.xStop := TRUE;
			Error.dwErrorActive := Error.dwErrorActive OR ERR_ROBOT_STOP;
			eState := E_ROBOT_STATE.ERROR;
		ELSIF xModbusError THEN
			Error.dwErrorActive := Error.dwErrorActive OR ERR_ROBOT_MODBUS_STUB;
			eState := E_ROBOT_STATE.ERROR;
		ELSIF xModbusDone THEN
			eState := E_ROBOT_STATE.DONE;
		END_IF;

    E_ROBOT_STATE.ERROR:

        Status.xBusy := FALSE;
        Status.xDone := FALSE;
        Status.xError := TRUE;

        IF xReset
        AND NOT Command.xExecute
        AND NOT Command.xStop
        AND NOT xGlobalError
        AND NOT stMotionManager.Status.xError
		AND NOT fbGripper.Status.xError
		AND NOT xModbusError THEN

			Error.dwErrorLast := Error.dwErrorActive;
            Error.dwErrorActive := DWORD#0;
            Status.xError := FALSE;
            eActiveAction := E_ROBOT_ACTION.NONE;
            eState := E_ROBOT_STATE.IDLE;
        END_IF;

END_CASE;

// =====================================================
// Формирование команды FB_MOTION_MANAGER
// =====================================================

stMotionManager.Command.xExecute := xMotionExecute;
stMotionManager.Command.eTargetPoint := eActivePoint;
stMotionManager.Command.xReset := xReset;

// В ST_MOTION_MANAGER_COMMAND нет отдельного xStop.
// Поэтому Stop передаётся как ошибка верхнего уровня.
stMotionManager.Command.xGlobalError :=
    xGlobalError OR Command.xStop;

// =====================================================
// Вызов FB_MOTION_MANAGER
// =====================================================

fbMotionManager(
    stPoint := stPoint,
    xReset := xReset,
    stMotionManager := stMotionManager,
    GroupData := GroupData,
    stPointManager := stPointManager
);

// =====================================================
// Вызов FB_GRIPPER
// =====================================================

stGripperCommand.xExecute := xGripperExecute;
stGripperCommand.xReset := xReset;
stGripperCommand.eAction := eActiveAction;

fbGripper(Command := stGripperCommand);

// =====================================================
// Общие статусы
// =====================================================

Status.eCurrentPoint := stMotionManager.Status.eCurrentPoint;
Status.xGripper1Open :=
    fbGripper.Status.xGripper1Open;

Status.xGripper1Closed :=
    fbGripper.Status.xGripper1Closed;

Status.xGripper2Open :=
    fbGripper.Status.xGripper2Open;

Status.xGripper2Closed :=
    fbGripper.Status.xGripper2Closed;

Status.xRotatedToBlank :=
    fbGripper.Status.xRotatedToBlank;

Status.xRotatedToDetail :=
    fbGripper.Status.xRotatedToDetail;

Status.xBlankAvailable := Status.xGripper1Closed;
Status.xDetailAvailable := Status.xGripper2Closed;

Diag.eState := eState;
Diag.eActiveAction := eActiveAction;
Diag.eActivePoint := eActivePoint;

IF Error.dwErrorActive <> DWORD#0 THEN
	Error.dwErrorLast := Error.dwErrorActive;
END_IF;

Error.stErrorActive := UpdateErrorView(dwError := Error.dwErrorActive);
Error.stErrorLast := UpdateErrorView(dwError := Error.dwErrorLast);

(* ---- FB_AXIS.UpdateErrorView.st ---- *)
METHOD UpdateErrorView : ST_AXIS_ERROR
VAR_INPUT
	dwAxisError   : DWORD; // Маска ошибок SoftMotion и привода
	dwLogicalError: DWORD; // Маска логических ошибок оси
END_VAR
VAR
	stError : ST_AXIS_ERROR; // Представление ошибок отдельными флагами
END_VAR

// --- BEGIN IMPLEMENTATION ---

stError.MC_POWER_ERROR := (dwAxisError AND AXE_MC_POWER_ERROR) <> DWORD#0;
stError.MC_RESET_ERROR := (dwAxisError AND AXE_MC_RESET_ERROR) <> DWORD#0;
stError.MC_STOP_ERROR := (dwAxisError AND AXE_MC_STOP_ERROR) <> DWORD#0;
stError.MC_JOG_ERROR := (dwAxisError AND AXE_MC_JOG_ERROR) <> DWORD#0;
stError.MC_HOME_ERROR := (dwAxisError AND AXE_MC_HOME_ERROR) <> DWORD#0;
stError.MC_MOVE_ABS_ERROR := (dwAxisError AND AXE_MC_MOVE_ABS_ERROR) <> DWORD#0;
stError.MC_MOVE_REL_ERROR := (dwAxisError AND AXE_MC_MOVE_REL_ERROR) <> DWORD#0;
stError.READ_POSITION_ERROR := (dwAxisError AND AXE_READ_POS_ERROR) <> DWORD#0;
stError.READ_STATUS_ERROR := (dwAxisError AND AXE_READ_STATUS_ERROR) <> DWORD#0;
stError.AXIS_ERRORSTOP := (dwAxisError AND AXE_ERRORSTOP) <> DWORD#0;
stError.FB_ERROR_OCCURRED := (dwAxisError AND AXE_FB_ERROR_OCCURRED) <> DWORD#0;
stError.COMMAND_ABORTED := (dwAxisError AND AXE_COMMAND_ABORTED) <> DWORD#0;
stError.UNKNOWN_AXIS_ERROR := (dwAxisError AND AXE_UNKNOWN_ACTUAL_ERROR) <> DWORD#0;
stError.DRIVE_AXIS_ERROR := (dwAxisError AND AXE_DRIVE_AXIS_ERROR) <> DWORD#0;

stError.POWER_PERMIT_LOST := (dwLogicalError AND LOG_POWER_PERMIT_LOST) <> DWORD#0;
stError.GLOBAL_DURING_POWER := (dwLogicalError AND LOG_GLOBAL_DURING_POWER) <> DWORD#0;
stError.GLOBAL_DURING_READY := (dwLogicalError AND LOG_GLOBAL_DURING_READY) <> DWORD#0;
stError.GLOBAL_DURING_MOTION := (dwLogicalError AND LOG_GLOBAL_DURING_MOTION) <> DWORD#0;
stError.JOG_CONFLICT := (dwLogicalError AND LOG_JOG_CONFLICT) <> DWORD#0;
stError.MOVE_ABS_NOT_HOMED := (dwLogicalError AND LOG_MOVE_ABS_NOT_HOMED) <> DWORD#0;
stError.MOVE_REL_NOT_HOMED := (dwLogicalError AND LOG_MOVE_REL_NOT_HOMED) <> DWORD#0;
stError.STEP_TIMEOUT := (dwLogicalError AND LOG_STEP_TIMEOUT) <> DWORD#0;
stError.UNKNOWN_STEP := (dwLogicalError AND LOG_UNKNOWN_STEP) <> DWORD#0;

UpdateErrorView := stError;

(* ---- FB_AXIS_GROUP.UpdateErrorView.st ---- *)
METHOD UpdateErrorView : ST_AXIS_GROUP_ERROR
VAR_INPUT
	dwMotionError : DWORD; // Маска ошибок блоков SoftMotion
	dwLogicalError: DWORD; // Маска логических ошибок группы
END_VAR
VAR
	stError : ST_AXIS_GROUP_ERROR; // Представление ошибок отдельными флагами
END_VAR

// --- BEGIN IMPLEMENTATION ---

stError.ENABLE_ERROR := (dwMotionError AND MOTION_ERR_ENABLE) <> DWORD#0;
stError.POWER_ERROR := (dwMotionError AND MOTION_ERR_POWER) <> DWORD#0;
stError.DISABLE_ERROR := (dwMotionError AND MOTION_ERR_DISABLE) <> DWORD#0;
stError.RESET_ERROR := (dwMotionError AND MOTION_ERR_RESET) <> DWORD#0;
stError.MOVE_DIRECT_ERROR := (dwMotionError AND MOTION_ERR_MOVE_DIRECT) <> DWORD#0;
stError.MOVE_LINEAR_ERROR := (dwMotionError AND MOTION_ERR_MOVE_LINEAR) <> DWORD#0;
stError.HALT_ERROR := (dwMotionError AND MOTION_ERR_HALT) <> DWORD#0;
stError.STOP_ERROR := (dwMotionError AND MOTION_ERR_STOP) <> DWORD#0;
stError.READ_POSITION_ERROR := (dwMotionError AND MOTION_ERR_READ_POSITION) <> DWORD#0;
stError.READ_STATUS_ERROR := (dwMotionError AND MOTION_ERR_READ_STATUS) <> DWORD#0;

stError.STEP_TIMEOUT := (dwLogicalError AND LOG_STEP_TIMEOUT) <> DWORD#0;
stError.INVALID_STATE := (dwLogicalError AND LOG_INVALID_STATE) <> DWORD#0;
stError.POWER_PERMIT_READY := (dwLogicalError AND LOG_POWER_PERMIT_READY) <> DWORD#0;
stError.POWER_PERMIT_LOST := (dwLogicalError AND LOG_POWER_PERMIT_LOST_DIRECT) <> DWORD#0;

UpdateErrorView := stError;

(* ---- FB_HMI.UpdateErrorView.st ---- *)
METHOD UpdateErrorView : ST_HMI_ERROR
VAR_INPUT
	dwError : DWORD; // Битовая маска для расшифровки
END_VAR
VAR
	stError : ST_HMI_ERROR; // Представление ошибок отдельными флагами
END_VAR

// --- BEGIN IMPLEMENTATION ---

stError.INTERNAL_ERROR := (dwError AND ERR_INTERNAL) <> DWORD#0;

UpdateErrorView := stError;

(* ---- FB_MACHINE.UpdateErrorView.st ---- *)
METHOD UpdateErrorView : ST_MACHINE_ERROR
VAR_INPUT
	dwError : DWORD; // Битовая маска для расшифровки
END_VAR
VAR
	stError : ST_MACHINE_ERROR; // Представление ошибок отдельными флагами
END_VAR

// --- BEGIN IMPLEMENTATION ---

stError.WRONG_OPERATION := (dwError AND ERR_WRONG_OPERATION) <> DWORD#0;
stError.WRONG_COMMAND := (dwError AND ERR_WRONG_COMMAND) <> DWORD#0;
stError.ROBOT_MOTION := (dwError AND ERR_ROBOT_MOTION) <> DWORD#0;
stError.ROBOT_ACTION := (dwError AND ERR_ROBOT_ACTION) <> DWORD#0;
stError.DOOR_OPEN := (dwError AND ERR_DOOR_OPEN) <> DWORD#0;
stError.DOOR_CLOSE := (dwError AND ERR_DOOR_CLOSE) <> DWORD#0;
stError.CHUCK_OPEN := (dwError AND ERR_CHUCK_OPEN) <> DWORD#0;
stError.CHUCK_CLOSE := (dwError AND ERR_CHUCK_CLOSE) <> DWORD#0;
stError.CYCLE_START := (dwError AND ERR_CYCLE_START) <> DWORD#0;
stError.SAFETY_STOP := (dwError AND ERR_SAFETY_STOP) <> DWORD#0;
stError.UNKNOWN_DETAIL := (dwError AND ERR_UNKNOWN_DETAIL) <> DWORD#0;
stError.MACHINE_ALARM := (dwError AND ERR_MACHINE_ALARM) <> DWORD#0;
stError.INDEX_ERROR := (dwError AND ERR_INDEX) <> DWORD#0;
stError.DOOR_ROBOT := (dwError AND ERR_DOOR_ROBOT) <> DWORD#0;
stError.MACHINE_IDLE := (dwError AND ERR_MACHINE_IDLE) <> DWORD#0;

UpdateErrorView := stError;

(* ---- FB_MACHINE_SIMULATION.UpdateErrorView.st ---- *)
METHOD UpdateErrorView : ST_MACHINE_SIM_ERROR
VAR_INPUT
	dwError : DWORD; // Битовая маска для расшифровки
END_VAR
VAR
	stError : ST_MACHINE_SIM_ERROR; // Представление ошибок отдельными флагами
END_VAR

// --- BEGIN IMPLEMENTATION ---

stError.MACHINE_ALARM := (dwError AND ERR_MACHINE_ALARM) <> DWORD#0;
stError.DOOR_FAULT := (dwError AND ERR_DOOR_FAULT) <> DWORD#0;
stError.CHUCK_FAULT := (dwError AND ERR_CHUCK_FAULT) <> DWORD#0;

UpdateErrorView := stError;

(* ---- FB_MAGAZINE.FIND_BLANK.st ---- *)
METHOD FIND_BLANK : SINT
VAR_INPUT
	iSlotCount : SINT; // Число слотов, участвующих в поиске
END_VAR
VAR_IN_OUT
	stDetail : ARRAY [1..GVL_CELL_SETTINGS.NumberDetail] OF ST_DETAIL; // Содержимое слотов магазина
END_VAR
VAR
	i : SINT; // Индекс проверяемого слота
END_VAR

// --- BEGIN IMPLEMENTATION ---

FIND_BLANK := 0;

FOR i:= 1 TO iSlotCount DO
	IF stDetail[i].xInPosition = TRUE AND stDetail[i].eDetailType =  E_DETAIL_TYPE.BLANK THEN
		FIND_BLANK := i;
		EXIT;
	END_IF
END_FOR

(* ---- FB_MAGAZINE.FIND_FREE_SLOT.st ---- *)
METHOD FIND_FREE_SLOT : SINT
VAR_INPUT
	iSlotCount : SINT; // Число слотов, участвующих в поиске
END_VAR
VAR_IN_OUT
	stDetail : ARRAY [1..GVL_CELL_SETTINGS.NumberDetail] OF ST_DETAIL; // Содержимое слотов магазина
END_VAR
VAR
	i : SINT; // Индекс проверяемого слота
END_VAR

// --- BEGIN IMPLEMENTATION ---

FIND_FREE_SLOT := 0;

FOR i:= 1 TO iSlotCount DO
	IF stDetail[i].xInPosition = FALSE THEN
		FIND_FREE_SLOT := i;
		EXIT;
	END_IF
END_FOR

(* ---- FB_MAGAZINE.UpdateErrorView.st ---- *)
METHOD UpdateErrorView : ST_MAGAZINE_ERROR
VAR_INPUT
	dwError : DWORD; // Битовая маска для расшифровки
END_VAR
VAR
	stError : ST_MAGAZINE_ERROR; // Представление ошибок отдельными флагами
END_VAR

// --- BEGIN IMPLEMENTATION ---

stError.WRONG_OPERATION := (dwError AND ERR_WRONG_OPERATION) <> DWORD#0;
stError.NO_BLANK := (dwError AND ERR_NO_BLANK) <> DWORD#0;
stError.NO_FREE_SLOT := (dwError AND ERR_NO_FREE_SLOT) <> DWORD#0;
stError.INVALID_SLOT := (dwError AND ERR_INVALID_SLOT) <> DWORD#0;
stError.SLOT_CONTENT := (dwError AND ERR_SLOT_CONTENT) <> DWORD#0;
stError.ROBOT_ERROR := (dwError AND ERR_ROBOT) <> DWORD#0;
stError.GLOBAL_STOP := (dwError AND ERR_GLOBAL_STOP) <> DWORD#0;
stError.GEOMETRY_ERROR := (dwError AND ERR_GEOMETRY) <> DWORD#0;

UpdateErrorView := stError;

(* ---- FB_POINT_MANAGER.UpdateErrorView.st ---- *)
METHOD UpdateErrorView : ST_POINT_MANAGER_ERROR
VAR_INPUT
	dwError : DWORD;
END_VAR
VAR
	stError: ST_POINT_MANAGER_ERROR;
END_VAR
// --- BEGIN IMPLEMENTATION ---

stError.X_OUT_OF_LIMIT    := (dwError AND X_OUT_OF_LIMIT ) <> 0;
stError.Y_OUT_OF_LIMIT := (dwError AND Y_OUT_OF_LIMIT ) <> 0;
stError.Z_OUT_OF_LIMIT := (dwError AND Z_OUT_OF_LIMIT ) <> 0;
stError.INVALID_VEL    := (dwError AND INVALID_VEL ) <> 0;

UpdateErrorView := stError;

(* ---- PLC_PRG.IsHmiCommandFresh.st ---- *)
METHOD PRIVATE IsHmiCommandFresh : BOOL
VAR_INPUT
	udiIssuedAtMs : UDINT;
END_VAR
VAR
	uliAgeMs : ULINT;
END_VAR

// --- BEGIN IMPLEMENTATION ---

// Explicit modulo-2^32 age: TIME() rolls over after about 49 days.
IF udiHmiCommandNowMs >= udiIssuedAtMs THEN
	uliAgeMs := UDINT_TO_ULINT(udiHmiCommandNowMs) - UDINT_TO_ULINT(udiIssuedAtMs);
ELSE
	uliAgeMs := ULINT#4294967296 + UDINT_TO_ULINT(udiHmiCommandNowMs) - UDINT_TO_ULINT(udiIssuedAtMs);
END_IF;
IsHmiCommandFresh := uliAgeMs <= UDINT_TO_ULINT(
	TIME_TO_UDINT(GVL_CELL_SETTINGS.tHmiCommandFreshnessTimeout)
);

(* ---- PLC_PRG.PublishHmi.st ---- *)
METHOD PRIVATE PublishHmi

// --- BEGIN IMPLEMENTATION ---

// Единый снимок состояния для внешней визуализации.
GVL_HMI.udiPlcHeartbeat := GVL_HMI.udiPlcHeartbeat + 1;
GVL_HMI.xHmiConnectionAlive := xHmiConnectionAlive;
GVL_HMI.xManualRecoveryActive := xManualRecoveryActive;
GVL_HMI.xGlobalError := GVL_CELL_CONTROL.xGlobalError;
GVL_HMI.xCellManual := GVL_CELL_CONTROL.xManual;
// Отказ тоже потребляет транзакцию: она не исполнится позже сама собой.
GVL_HMI.udiCellModeAckSeq := udiCellModeCommandSnapshot;
GVL_HMI.xErrorSimulationEnabled := GVL_CELL_SETTINGS.xErrorSimulationEnabled;
GVL_HMI.stSafetyFaultStatus := CELL_SAFETY.FaultStatus;
GVL_HMI.xSimulationAccelerationActive := GVL_CELL_SETTINGS.xSimulationAccelerationActive;
GVL_HMI.xSimulationAccelerationChangeAllowed := GVL_CELL_SETTINGS.xSimulationAccelerationChangeAllowed;
GVL_HMI.uiSimulationTimeFactorApplied := GVL_CELL_SETTINGS.uiSimulationTimeFactorApplied;
GVL_HMI.xSimulationAccelerationPending := GVL_CELL_SETTINGS.xSimulationAccelerationPending;
GVL_HMI.xSimulationAccelerationBusy := GVL_CELL_SETTINGS.xSimulationAccelerationBusy;
GVL_HMI.xSimulationAccelerationError := GVL_CELL_SETTINGS.xSimulationAccelerationError;
GVL_HMI.udiSimulationAccelerationErrorId := GVL_CELL_SETTINGS.udiSimulationAccelerationErrorId;
GVL_HMI.lrSafetyHomeX := GVL_POINT.Points[E_POINT_NAME.HOME_SAFETY].X;
GVL_HMI.lrSafetyHomeY := GVL_POINT.Points[E_POINT_NAME.HOME_SAFETY].Y;
GVL_HMI.lrSafetyHomeZ := GVL_POINT.Points[E_POINT_NAME.HOME_SAFETY].Z;
GVL_HMI.lrSafetyHomeSpeedFactor := GVL_POINT.Points[E_POINT_NAME.HOME_SAFETY].SpeedFactor;
GVL_HMI.lrSafetyHomeToleranceX := GVL_CELL_SETTINGS.lrSafetyHomeToleranceX;
GVL_HMI.lrSafetyHomeToleranceY := GVL_CELL_SETTINGS.lrSafetyHomeToleranceY;
GVL_HMI.lrSafetyHomeToleranceZ := GVL_CELL_SETTINGS.lrSafetyHomeToleranceZ;
GVL_HMI.rRobotAccelerationPercent := GVL_CELL_SETTINGS.rRobotAccelerationPercent;
GVL_HMI.rRobotDecelerationPercent := GVL_CELL_SETTINGS.rRobotDecelerationPercent;
GVL_HMI.rRobotJerkPercent := GVL_CELL_SETTINGS.rRobotJerkPercent;
GVL_HMI.lrRobotHaltDeceleration := GVL_CELL_SETTINGS.lrRobotHaltDeceleration;
GVL_HMI.lrRobotHaltJerk := GVL_CELL_SETTINGS.lrRobotHaltJerk;
GVL_HMI.stCellMachineTimeouts := GVL_CELL_SETTINGS.stMachineTimeouts;
GVL_HMI.stCellAxisTimeouts := GVL_CELL_SETTINGS.stAxisTimeouts;
GVL_HMI.stCellAxisGroupTimeouts := GVL_CELL_SETTINGS.stAxisGroupTimeouts;
GVL_HMI.tPointCheckStartTimeout := GVL_CELL_SETTINGS.tPointCheckStartTimeout;
GVL_HMI.tSimulationDynamicsTimeout := GVL_CELL_SETTINGS.tSimulationDynamicsTimeout;
GVL_HMI.tHmiWatchdogTimeout := GVL_CELL_SETTINGS.tHmiWatchdogTimeout;
GVL_HMI.tMobileMotionWatchdogTimeout := GVL_CELL_SETTINGS.tMobileMotionWatchdogTimeout;
GVL_HMI.tPointCheckWatchdogTimeout := GVL_CELL_SETTINGS.tPointCheckWatchdogTimeout;
GVL_HMI.tHmiCommandFreshnessTimeout := GVL_CELL_SETTINGS.tHmiCommandFreshnessTimeout;
GVL_HMI.xCellSettingsChangeAllowed := GVL_CELL_SETTINGS.xCellSettingsChangeAllowed;
GVL_HMI.rPointCheckSpeedPercent := GVL_CELL_SETTINGS.rPointCheckSpeedPercent;
GVL_HMI.xPointCheckActive := xPointCheckActive;
IF xPointCheckActive THEN
	GVL_HMI.rPointCheckAppliedSpeedPercent := rPointCheckLatchedSpeed;
ELSE
	GVL_HMI.rPointCheckAppliedSpeedPercent := GVL_CELL_SETTINGS.rPointCheckSpeedPercent;
END_IF;
GVL_HMI.xPointTableReady := xPointTableReady;
GVL_HMI.astPointEditorPoints[1] := GVL_POINT.Points[E_POINT_NAME.MACHINE_1_ABOVE];
GVL_HMI.astPointEditorPoints[2] := GVL_POINT.Points[E_POINT_NAME.MACHINE_1_CHUCK_APROACH];
GVL_HMI.astPointEditorPoints[3] := GVL_POINT.Points[E_POINT_NAME.MACHINE_1_CHUCK_POSITION];
GVL_HMI.astPointEditorPoints[4] := GVL_POINT.Points[E_POINT_NAME.MACHINE_2_ABOVE];
GVL_HMI.astPointEditorPoints[5] := GVL_POINT.Points[E_POINT_NAME.MACHINE_2_CHUCK_APROACH];
GVL_HMI.astPointEditorPoints[6] := GVL_POINT.Points[E_POINT_NAME.MACHINE_2_CHUCK_POSITION];
GVL_HMI.astPointEditorPoints[7] := GVL_POINT.Points[E_POINT_NAME.MACHINE_3_ABOVE];
GVL_HMI.astPointEditorPoints[8] := GVL_POINT.Points[E_POINT_NAME.MACHINE_3_CHUCK_APROACH];
GVL_HMI.astPointEditorPoints[9] := GVL_POINT.Points[E_POINT_NAME.MACHINE_3_CHUCK_POSITION];
GVL_HMI.astPointEditorPoints[10] := GVL_POINT.Points[E_POINT_NAME.HOME_SAFETY];
GVL_HMI.astPointEditorPoints[11] := GVL_POINT.Points[E_POINT_NAME.MAGAZINE_1_DETAIL];
GVL_HMI.astPointEditorPoints[12] := GVL_POINT.Points[E_POINT_NAME.MAGAZINE_2_DETAIL];
GVL_HMI.auiPointEditorPointId[1] := TO_UINT(E_POINT_NAME.MACHINE_1_ABOVE);
GVL_HMI.auiPointEditorPointId[2] := TO_UINT(E_POINT_NAME.MACHINE_1_CHUCK_APROACH);
GVL_HMI.auiPointEditorPointId[3] := TO_UINT(E_POINT_NAME.MACHINE_1_CHUCK_POSITION);
GVL_HMI.auiPointEditorPointId[4] := TO_UINT(E_POINT_NAME.MACHINE_2_ABOVE);
GVL_HMI.auiPointEditorPointId[5] := TO_UINT(E_POINT_NAME.MACHINE_2_CHUCK_APROACH);
GVL_HMI.auiPointEditorPointId[6] := TO_UINT(E_POINT_NAME.MACHINE_2_CHUCK_POSITION);
GVL_HMI.auiPointEditorPointId[7] := TO_UINT(E_POINT_NAME.MACHINE_3_ABOVE);
GVL_HMI.auiPointEditorPointId[8] := TO_UINT(E_POINT_NAME.MACHINE_3_CHUCK_APROACH);
GVL_HMI.auiPointEditorPointId[9] := TO_UINT(E_POINT_NAME.MACHINE_3_CHUCK_POSITION);
GVL_HMI.auiPointEditorPointId[10] := TO_UINT(E_POINT_NAME.HOME_SAFETY);
GVL_HMI.auiPointEditorPointId[11] := TO_UINT(E_POINT_NAME.MAGAZINE_1_DETAIL);
GVL_HMI.auiPointEditorPointId[12] := TO_UINT(E_POINT_NAME.MAGAZINE_2_DETAIL);
GVL_HMI.xModbusMode := GVL_ROBOT_MODBUS.xModeActive;
GVL_HMI.xRobotModeChangeAllowed := GVL_ROBOT_MODBUS.xRobotModeChangeAllowed;
GVL_HMI.xModbusSettingsChangeAllowed := GVL_ROBOT_MODBUS.xSettingsChangeAllowed;
GVL_HMI.stRobotModbusStatus := GVL_ROBOT_MODBUS.Status;
uiMagazine := GVL_CELL_MANAGER.Status.uiActiveMagazine;
IF (uiMagazine < UINT#1) OR (uiMagazine > UINT#2) THEN
	uiMagazine := UINT#1;
END_IF;
GVL_HMI.stTestObservability.udiAppliedScenarioSeq := GVL_HMI.udiTestScenarioAckSeq;
GVL_HMI.stTestObservability.uiCellState := TO_UINT(GVL_CELL_MANAGER.Diag.eState);
GVL_HMI.stTestObservability.uiRobotState := TO_UINT(GVL_ROBOT.Diag.eState);
GVL_HMI.stTestObservability.uiRobotAction := TO_UINT(GVL_ROBOT.Diag.eActiveAction);
GVL_HMI.stTestObservability.uiRobotPoint := TO_UINT(GVL_ROBOT.Diag.eActivePoint);
GVL_HMI.stTestObservability.uiActiveMagazine := GVL_CELL_MANAGER.Status.uiActiveMagazine;
GVL_HMI.stTestObservability.uiMagazineState := TO_UINT(GVL_MAGAZINE.astDiag[uiMagazine].eState);
GVL_HMI.stTestObservability.uiMagazineOperation := TO_UINT(GVL_MAGAZINE.astStatus[uiMagazine].eActualOperation);
GVL_HMI.stTestObservability.uiTakeSlot := SINT_TO_UINT(GVL_MAGAZINE.astStatus[uiMagazine].iSelectedBlank);
GVL_HMI.stTestObservability.uiPutSlot := SINT_TO_UINT(GVL_MAGAZINE.astStatus[uiMagazine].iSelectedFreeSlot);
GVL_HMI.stTestObservability.uiSelectedMachine := GVL_CELL_MANAGER.Status.uiSelectedMachine;
GVL_HMI.stTestObservability.uiSelectedType := GVL_MULTI_TYPE.CycleStatus.uiSelectedType;
GVL_HMI.stTestObservability.uiErrorSource := UINT#0;
GVL_HMI.stTestObservability.dwErrorCode := DWORD#0;
FOR uiMachine := 1 TO 3 DO
	GVL_HMI.stTestObservability.auiMachineState[uiMachine] := TO_UINT(GVL_MACHINE.Diag[uiMachine].eState);
	GVL_HMI.stTestObservability.auiMachineOperation[uiMachine] := TO_UINT(GVL_MACHINE.Diag[uiMachine].eActualOperation);
END_FOR;
IF GVL_ROBOT.Error.dwErrorActive <> DWORD#0 THEN
	GVL_HMI.stTestObservability.uiErrorSource := UINT#2;
	GVL_HMI.stTestObservability.dwErrorCode := GVL_ROBOT.Error.dwErrorActive;
ELSIF GVL_MAGAZINE.astError[1].dwErrorActive <> DWORD#0 THEN
	GVL_HMI.stTestObservability.uiErrorSource := UINT#3;
GVL_HMI.stTestObservability.dwErrorCode := GVL_MAGAZINE.astError[1].dwErrorActive;
ELSIF GVL_MAGAZINE.astError[2].dwErrorActive <> DWORD#0 THEN
	GVL_HMI.stTestObservability.uiErrorSource := UINT#7;
	GVL_HMI.stTestObservability.dwErrorCode := GVL_MAGAZINE.astError[2].dwErrorActive;
ELSIF GVL_CELL_MANAGER.Error.dwErrorActive <> DWORD#0 THEN
	GVL_HMI.stTestObservability.uiErrorSource := UINT#1;
	GVL_HMI.stTestObservability.dwErrorCode := GVL_CELL_MANAGER.Error.dwErrorActive;
ELSE
	FOR uiMachine := 1 TO 3 DO
		IF GVL_MACHINE.Error[uiMachine].dwErrorActive <> DWORD#0 THEN
			GVL_HMI.stTestObservability.uiErrorSource := uiMachine + UINT#3;
			GVL_HMI.stTestObservability.dwErrorCode := GVL_MACHINE.Error[uiMachine].dwErrorActive;
		END_IF;
	END_FOR;
END_IF;
FOR uiMachine := 1 TO 9 DO
	GVL_HMI.auiRobotModbusWriteRegisters[uiMachine] :=
		GVL_ROBOT_MODBUS.auiWriteRegisters[uiMachine - 1];
END_FOR;
FOR uiMachine := 1 TO 17 DO
	GVL_HMI.auiRobotModbusReadRegisters[uiMachine] :=
		GVL_ROBOT_MODBUS.auiReadRegisters[uiMachine - 1];
END_FOR;
GVL_HMI.xSimAxisGroupErrorAllowed := GVL_AXIS_GROUP.AxisGroup.Status.xSimErrorAllowed;
GVL_HMI.astAxisFaultStatus[1] := AXIS_X.FaultStatus;
GVL_HMI.astAxisFaultStatus[2] := AXIS_Y.FaultStatus;
GVL_HMI.astAxisFaultStatus[3] := AXIS_Z.FaultStatus;
GVL_HMI.stAxisGroupFaultStatus := GROUP_XYZ.FaultStatus;
GVL_HMI.stGripperFaultStatus := ROBOT.FaultStatus.stGripper;
GVL_HMI.stRobotFaultStatus := ROBOT.FaultStatus.stRobot;
GVL_HMI.stCellFaultStatus := CELL_MANAGER.FaultStatus;
GVL_HMI.stPointFaultStatus := ROBOT.FaultStatus.stPoint;
GVL_HMI.stMagazineFaultStatus := fbMagazine1.FaultStatus;
GVL_HMI.astMagazineFaultStatus[1] := fbMagazine1.FaultStatus;
GVL_HMI.astMagazineFaultStatus[2] := fbMagazine2.FaultStatus;
GVL_HMI.rLoadCNC_1 := GVL_STATISTIC.stStatistic.stMachineStat.rLoadCNC_1;
GVL_HMI.rLoadCNC_2 := GVL_STATISTIC.stStatistic.stMachineStat.rLoadCNC_2;
GVL_HMI.rLoadCNC_3 := GVL_STATISTIC.stStatistic.stMachineStat.rLoadCNC_3;
GVL_HMI.rRobot := GVL_STATISTIC.stStatistic.stRobotStat.rRobot;

GVL_HMI.stCellStatus := GVL_CELL_MANAGER.Status;
GVL_HMI.stCellStatus.xResetAllowed := xAlarmResetAllowed;
GVL_HMI.stCellDiag := GVL_CELL_MANAGER.Diag;
GVL_HMI.stCellError := GVL_CELL_MANAGER.Error;
GVL_HMI.stCellSafetyStatus := CELL_SAFETY.Status;
GVL_HMI.stCellSafetyDiag := CELL_SAFETY.Diag;
GVL_HMI.stCellSafetyError := CELL_SAFETY.Error;
GVL_HMI.astButtonStationIoStatus := CELL_SAFETY.astButtonStationIoStatus;
GVL_HMI.stFrontControlCabinetIoStatus := CELL_SAFETY.stFrontControlCabinetIoStatus;
GVL_HMI.xSignalTowerRed := GVL_CELL_SAFETY_IO.xSignalTowerRedOutput;
GVL_HMI.xSignalTowerAmber := GVL_CELL_SAFETY_IO.xSignalTowerAmberOutput;
GVL_HMI.xSignalTowerGreen := GVL_CELL_SAFETY_IO.xSignalTowerGreenOutput;
GVL_HMI.stRearControlCabinetIoStatus := CELL_SAFETY.stRearControlCabinetIoStatus;
GVL_HMI.stMpgIoStatus := CELL_SAFETY.stMpgIoStatus;
GVL_HMI.astEnclosureDoorStatus := CELL_SAFETY.astEnclosureDoorStatus;
GVL_HMI.stMultiType.Config := GVL_MULTI_TYPE.Config;
GVL_HMI.stMultiType.ConfigStatus := GVL_MULTI_TYPE.ConfigStatus;
GVL_HMI.stMultiType.CycleStatus := GVL_MULTI_TYPE.CycleStatus;

GVL_HMI.stRobotStatus := GVL_ROBOT.Status;
GVL_HMI.stRobotDiag := GVL_ROBOT.Diag;
GVL_HMI.stRobotError := GVL_ROBOT.Error;
GVL_HMI.stGripperDiag := GVL_ROBOT.GripperDiag;
GVL_HMI.stGripperError := GVL_ROBOT.GripperError;
GVL_HMI.stAxisGroupStatus := GVL_AXIS_GROUP.AxisGroup.Status;
GVL_HMI.stAxisGroupDiag := GVL_AXIS_GROUP.AxisGroup.Diag;
GVL_HMI.stAxisGroupError := GVL_AXIS_GROUP.AxisGroup.Error;
GVL_HMI.stMotionManagerStatus := GVL_MOTION_MANAGER.stMotionManager.Status;
GVL_HMI.stMotionManagerDiag := GVL_MOTION_MANAGER.stMotionManager.Diag;
GVL_HMI.stMotionManagerError := GVL_MOTION_MANAGER.stMotionManager.Error;
GVL_HMI.stPointManagerStatus := GVL_POINT_MANAGER.PointManager.Status;
GVL_HMI.stPointManagerDiag := GVL_POINT_MANAGER.PointManager.Diag;
GVL_HMI.stPointManagerError := GVL_POINT_MANAGER.PointManager.Error;

FOR uiMachine := 1 TO 3 DO
	GVL_HMI.astAxisStatus[uiMachine] := GVL_AXIS.arrAxis[uiMachine].Status;
	GVL_HMI.astAxisDiag[uiMachine] := GVL_AXIS.arrAxis[uiMachine].Diag;
	GVL_HMI.astAxisError[uiMachine] := GVL_AXIS.arrAxis[uiMachine].Error;
END_FOR;

GVL_HMI.stMagazineStatus := GVL_MAGAZINE.astStatus[1];
GVL_HMI.stMagazineDiag := GVL_MAGAZINE.astDiag[1];
GVL_HMI.stMagazineError := GVL_MAGAZINE.astError[1];
FOR uiMagazine := UINT#1 TO UINT#2 DO
	GVL_HMI.astMagazineStatus[uiMagazine] := GVL_MAGAZINE.astStatus[uiMagazine];
	GVL_HMI.astMagazineDiag[uiMagazine] := GVL_MAGAZINE.astDiag[uiMagazine];
	GVL_HMI.astMagazineError[uiMagazine] := GVL_MAGAZINE.astError[uiMagazine];
	GVL_HMI.astMagazineInventory[uiMagazine] := GVL_DETAIL.astMagazine[uiMagazine];
END_FOR;
GVL_HMI.stAlarmStatus := GVL_ALARM.Status;
GVL_HMI.astAlarmEvent := GVL_ALARM.Events;

FOR uiMachine := 1 TO 3 DO
	GVL_HMI.astMachineStatus[uiMachine] := GVL_MACHINE.Status[uiMachine];
	GVL_HMI.astMachineDiag[uiMachine] := GVL_MACHINE.Diag[uiMachine];
	GVL_HMI.astMachineError[uiMachine] := GVL_MACHINE.Error[uiMachine];
	CASE uiMachine OF
		1:
			GVL_HMI.astMachineFaultStatus[uiMachine] := MACHINE_1_FAULT.Status;
			GVL_HMI.astMachineFaultStatus[uiMachine].xResetAllowed :=
				MACHINE_1_SIM.Diag.xResetAllowed OR GVL_MACHINE.Status[uiMachine].xResetAllowed;
		2:
			GVL_HMI.astMachineFaultStatus[uiMachine] := MACHINE_2_FAULT.Status;
			GVL_HMI.astMachineFaultStatus[uiMachine].xResetAllowed :=
				MACHINE_2_SIM.Diag.xResetAllowed OR GVL_MACHINE.Status[uiMachine].xResetAllowed;
		3:
			GVL_HMI.astMachineFaultStatus[uiMachine] := MACHINE_3_FAULT.Status;
			GVL_HMI.astMachineFaultStatus[uiMachine].xResetAllowed :=
				MACHINE_3_SIM.Diag.xResetAllowed OR GVL_MACHINE.Status[uiMachine].xResetAllowed;
	END_CASE;
END_FOR;

GVL_HMI.astMachineIoStatus[1] := MACHINE_1_FAULT.MachineStatus;
GVL_HMI.astMachineIoStatus[2] := MACHINE_2_FAULT.MachineStatus;
GVL_HMI.astMachineIoStatus[3] := MACHINE_3_FAULT.MachineStatus;
GVL_HMI.astMachineRawIoStatus[1] := MACHINE_1_SIM.Status;
GVL_HMI.astMachineRawIoStatus[2] := MACHINE_2_SIM.Status;
GVL_HMI.astMachineRawIoStatus[3] := MACHINE_3_SIM.Status;
GVL_HMI.astMachineTimeouts[1] := MACHINE_1_FAULT.Timeouts;
GVL_HMI.astMachineTimeouts[2] := MACHINE_2_FAULT.Timeouts;
GVL_HMI.astMachineTimeouts[3] := MACHINE_3_FAULT.Timeouts;
GVL_HMI.astMachineSimDiag[1] := MACHINE_1_SIM.Diag;
GVL_HMI.astMachineSimDiag[2] := MACHINE_2_SIM.Diag;
GVL_HMI.astMachineSimDiag[3] := MACHINE_3_SIM.Diag;
GVL_HMI.astMachineSimError[1] := MACHINE_1_SIM.Error;
GVL_HMI.astMachineSimError[2] := MACHINE_2_SIM.Error;
GVL_HMI.astMachineSimError[3] := MACHINE_3_SIM.Error;

FOR iDetail := 1 TO GVL_CELL_SETTINGS.NumberDetail DO
	GVL_HMI.astMagazineSlot[iDetail] := GVL_DETAIL.astMagazine[1].aSlots[iDetail];
END_FOR;

// Ack only the snapshot actually dispatched through all consumers this scan.
FOR uiHmiCommandIndex := UINT#1 TO UINT#121 DO
	IF axHmiCommandConsumed[uiHmiCommandIndex] THEN
		GVL_HMI.audiHmiCommandAckSeq[uiHmiCommandIndex] := audiHmiCommandSnapshot[uiHmiCommandIndex];
	END_IF;
END_FOR;
GVL_HMI.udiCellSettingAckSeq := udiCellSettingSnapshot;
